// ============================================
// DB_RecipeProgram1 - Program 1
// Lines: 500
// CHUNKS: 5 x 100
// Generated by SpinningCam  [2026-09-24 16:45:37]
// !!! CONTINUOUS MOTION (CMD=2) - EXPERIMENTAL PLC ONLY !!!
// Load ONLY on the continuous-motion PLC build. A production PLC
// skips CMD=2 lines and jumps straight between the other points.
// T=0.045 s, corner tol=0.2 mm, F min=180, exact stop at >= 90 deg, stop slow-down=OFF
// CMD=2 lines: 483, exact corners: 2, slowed corners: 1 (+1 leaving), slowed stops: 0
// ============================================
//
// --- MAKINE AYARLARI ---
// Machine Origin  : X=0.0, Z=0.0
// Axis Direction  : X=NORMAL, Z=NORMAL
// Output Mode     : RADIUS
// G54 Offset      : X=0.0, Z=0.0
// Home            : X=-394.0, Z=-174.0
// Retract         : X=-10.0, Z=-10.0
//
// --- PARCA / BLANK ---
// Blank Radius    : 150.0 mm
// Blank Z Shift   : 0.0 mm
// Final Thickness : 0.8 mm
// Min Safety Gap  : 0.0 mm
//
// --- MANDREL POZISYON ---
// Mandrel Offset  : X=0.0, Z=0.0
// Mandrel Rot     : Rx=90.0, Ry=0.0, Rz=0.0
//
// --- OPERASYONLAR ---
// Op1: ROUGHING, 1 paso, T004, R=44.56mm, RPM=600.0, mm_min=1000.0
// Op2: ROUGHING, 1 paso, T004, R=44.56mm, RPM=600.0, mm_min=1000.0
// Op3: ROUGHING, 1 paso, T004, R=44.56mm, RPM=600.0, mm_min=1000.0
// Op4: ROUGHING, 1 paso, T004, R=44.56mm, RPM=600.0, mm_min=1000.0
// Op5: ROUGHING, 1 paso, T004, R=44.56mm, RPM=600.0, mm_min=1000.0
// Op6: ROUGHING, 1 paso, T004, R=44.56mm, RPM=600.0, mm_min=1000.0
// Op7: ROUGHING, 1 paso, T004, R=44.56mm, RPM=600.0, mm_min=1000.0
// Op8: ROUGHING, 1 paso, T004, R=44.56mm, RPM=600.0, mm_min=1000.0
// Op9: ROUGHING, 1 paso, T004, R=44.56mm, RPM=600.0, mm_min=1000.0
// Op10: ROUGHING, 1 paso, T004, R=44.56mm, RPM=600.0, mm_min=1000.0
// Op11: ROUGHING, 1 paso, T004, R=44.56mm, RPM=600.0, mm_min=1000.0
// Op12: ROUGHING, 1 paso, T004, R=44.56mm, RPM=600.0, mm_min=1000.0
// Op13: ROUGHING, 1 paso, T004, R=44.56mm, RPM=600.0, mm_min=1000.0
// Op14: ROUGHING, 1 paso, T004, R=44.56mm, RPM=600.0, mm_min=1000.0
// Op15: ROUGHING, 1 paso, T004, R=44.56mm, RPM=600.0, mm_min=1000.0
// Op16: ROUGHING, 1 paso, T004, R=44.56mm, RPM=600.0, mm_min=1000.0
// Op17: ROUGHING, 1 paso, T004, R=44.56mm, RPM=600.0, mm_min=1000.0
// Op18: CUTTING, 1 paso, T006, R=5.0mm, RPM=500.0, mm_min=7.0
// Op19: ROUGHING, 1 paso, T004, R=44.56mm, RPM=600.0, mm_min=1000.0
// Op20: ROUGHING, 1 paso, T004, R=44.56mm, RPM=600.0, mm_min=1000.0
// Op21: ROUGHING, 1 paso, T004, R=44.56mm, RPM=600.0, mm_min=1000.0
// Op22: ROUGHING, 1 paso, T004, R=44.56mm, RPM=600.0, mm_min=1000.0
// Op23: ROUGHING, 1 paso, T004, R=44.56mm, RPM=600.0, mm_min=1000.0
// Op24: ROUGHING, 1 paso, T004, R=44.56mm, RPM=600.0, mm_min=1000.0
// Op25: ROUGHING, 1 paso, T004, R=44.56mm, RPM=600.0, mm_min=1000.0
// Op26: ROUGHING, 1 paso, T004, R=44.56mm, RPM=600.0, mm_min=1000.0
// Op27: ROUGHING, 1 paso, T004, R=44.56mm, RPM=600.0, mm_min=1000.0
// Op28: ROUGHING, 1 paso, T004, R=44.56mm, RPM=600.0, mm_min=1000.0
// Op29: ROUGHING, 1 paso, T004, R=44.56mm, RPM=600.0, mm_min=1000.0
// Op30: ROUGHING, 1 paso, T004, R=44.56mm, RPM=600.0, mm_min=1000.0
// Op31: ROUGHING, 1 paso, T004, R=44.56mm, RPM=600.0, mm_min=1000.0
// Op32: ROUGHING, 1 paso, T004, R=44.56mm, RPM=600.0, mm_min=1000.0
// Op33: ROUGHING, 1 paso, T004, R=44.56mm, RPM=600.0, mm_min=1000.0
// Op34: ROUGHING, 1 paso, T004, R=44.56mm, RPM=600.0, mm_min=1000.0
// Op35: ROUGHING, 1 paso, T004, R=44.56mm, RPM=600.0, mm_min=1000.0
// Op36: ROUGHING, 1 paso, T004, R=44.56mm, RPM=600.0, mm_min=1000.0
// Op37: ROUGHING, 1 paso, T004, R=44.56mm, RPM=600.0, mm_min=1000.0
// Op38: ROUGHING, 1 paso, T004, R=44.56mm, RPM=600.0, mm_min=1000.0
// Op39: ROUGHING, 1 paso, T004, R=44.56mm, RPM=600.0, mm_min=1000.0
// Op40: ROUGHING, 1 paso, T004, R=44.56mm, RPM=600.0, mm_min=1000.0
// Op41: ROUGHING, 1 paso, T004, R=44.56mm, RPM=600.0, mm_min=1000.0
// Op42: ROUGHING, 1 paso, T004, R=44.56mm, RPM=600.0, mm_min=1000.0
// Op43: ROUGHING, 1 paso, T004, R=44.56mm, RPM=600.0, mm_min=1000.0
// Op44: ROUGHING, 1 paso, T004, R=44.56mm, RPM=600.0, mm_min=1000.0
// Op45: ROUGHING, 1 paso, T004, R=44.56mm, RPM=600.0, mm_min=1000.0
// Op46: ROUGHING, 1 paso, T004, R=44.56mm, RPM=600.0, mm_min=1000.0
// Op47: ROUGHING, 1 paso, T004, R=44.56mm, RPM=600.0, mm_min=1000.0
// Op48: ROUGHING, 1 paso, T004, R=44.56mm, RPM=600.0, mm_min=1000.0
// Op49: ROUGHING, 1 paso, T004, R=44.56mm, RPM=600.0, mm_min=1000.0
// Op50: ROUGHING, 1 paso, T004, R=44.56mm, RPM=600.0, mm_min=1000.0
// Op51: ROUGHING, 1 paso, T004, R=44.56mm, RPM=600.0, mm_min=1000.0
// Op52: ROUGHING, 1 paso, T004, R=44.56mm, RPM=600.0, mm_min=1000.0
// Op53: ROUGHING, 1 paso, T004, R=44.56mm, RPM=600.0, mm_min=1000.0
// Op54: ROUGHING, 1 paso, T004, R=44.56mm, RPM=600.0, mm_min=1000.0
// Op55: ROUGHING, 1 paso, T004, R=44.56mm, RPM=600.0, mm_min=1000.0
// Op56: ROUGHING, 1 paso, T004, R=44.56mm, RPM=600.0, mm_min=1000.0
// Op57: ROUGHING, 1 paso, T004, R=44.56mm, RPM=600.0, mm_min=1000.0
// Op58: ROUGHING, 1 paso, T004, R=44.56mm, RPM=600.0, mm_min=1000.0
// Op59: ROUGHING, 1 paso, T004, R=44.56mm, RPM=600.0, mm_min=1000.0
// Op60: ROUGHING, 1 paso, T004, R=44.56mm, RPM=600.0, mm_min=1000.0
// Op61: ROUGHING, 1 paso, T004, R=44.56mm, RPM=600.0, mm_min=1000.0
// Op62: ROUGHING, 1 paso, T004, R=44.56mm, RPM=600.0, mm_min=1000.0
// Op63: ROUGHING, 1 paso, T004, R=44.56mm, RPM=600.0, mm_min=1000.0
// Op64: ROUGHING, 1 paso, T004, R=44.56mm, RPM=600.0, mm_min=1000.0
// Op65: ROUGHING, 1 paso, T004, R=44.56mm, RPM=600.0, mm_min=1000.0
// Op66: ROUGHING, 1 paso, T004, R=44.56mm, RPM=600.0, mm_min=1000.0
// Op67: ROUGHING, 1 paso, T004, R=44.56mm, RPM=600.0, mm_min=1000.0
// Op68: ROUGHING, 1 paso, T004, R=44.56mm, RPM=600.0, mm_min=1000.0
// Op69: ROUGHING, 1 paso, T004, R=44.56mm, RPM=600.0, mm_min=1000.0
// Op70: ROUGHING, 1 paso, T004, R=44.56mm, RPM=600.0, mm_min=1000.0
// Op71: ROUGHING, 1 paso, T004, R=44.56mm, RPM=600.0, mm_min=1000.0
// Op72: ROUGHING, 1 paso, T004, R=44.56mm, RPM=600.0, mm_min=1000.0
// Op73: ROUGHING, 1 paso, T004, R=44.56mm, RPM=600.0, mm_min=1000.0
// Op74: ROUGHING, 1 paso, T004, R=44.56mm, RPM=600.0, mm_min=1000.0
// Op75: ROUGHING, 1 paso, T004, R=44.56mm, RPM=600.0, mm_min=1000.0
// Op76: ROUGHING, 1 paso, T004, R=44.56mm, RPM=600.0, mm_min=1000.0
// Op77: ROUGHING, 1 paso, T004, R=44.56mm, RPM=600.0, mm_min=1000.0
// Op78: ROUGHING, 1 paso, T004, R=44.56mm, RPM=600.0, mm_min=1000.0
// Op79: ROUGHING, 1 paso, T004, R=44.56mm, RPM=600.0, mm_min=1000.0
// Op80: ROUGHING, 1 paso, T004, R=44.56mm, RPM=600.0, mm_min=1000.0
// Op81: ROUGHING, 1 paso, T004, R=44.56mm, RPM=600.0, mm_min=1000.0
// Op82: ROUGHING, 1 paso, T004, R=44.56mm, RPM=600.0, mm_min=1000.0
// Op83: ROUGHING, 1 paso, T004, R=44.56mm, RPM=600.0, mm_min=1000.0
// Op84: ROUGHING, 1 paso, T004, R=44.56mm, RPM=600.0, mm_min=1000.0
// Op85: ROUGHING, 1 paso, T004, R=44.56mm, RPM=600.0, mm_min=1000.0
// Op86: ROUGHING, 1 paso, T004, R=44.56mm, RPM=600.0, mm_min=1000.0
// Op87: ROUGHING, 1 paso, T004, R=44.56mm, RPM=600.0, mm_min=1000.0
// Op88: ROUGHING, 1 paso, T004, R=44.56mm, RPM=600.0, mm_min=1000.0
// Op89: ROUGHING, 1 paso, T004, R=44.56mm, RPM=600.0, mm_min=1000.0
// Op90: ROUGHING, 1 paso, T004, R=44.56mm, RPM=600.0, mm_min=1000.0
// Op91: ROUGHING, 1 paso, T004, R=44.56mm, RPM=600.0, mm_min=1000.0
// Op92: ROUGHING, 1 paso, T004, R=44.56mm, RPM=600.0, mm_min=1000.0
// Op93: ROUGHING, 1 paso, T004, R=44.56mm, RPM=600.0, mm_min=1000.0
// Op94: ROUGHING, 1 paso, T004, R=44.56mm, RPM=600.0, mm_min=1000.0
// Op95: ROUGHING, 1 paso, T004, R=44.56mm, RPM=600.0, mm_min=1000.0
// Op96: ROUGHING, 1 paso, T004, R=44.56mm, RPM=600.0, mm_min=1000.0
// Op97: ROUGHING, 1 paso, T004, R=44.56mm, RPM=600.0, mm_min=1000.0
// Op98: ROUGHING, 1 paso, T004, R=44.56mm, RPM=600.0, mm_min=1000.0
// Op99: ROUGHING, 1 paso, T004, R=44.56mm, RPM=600.0, mm_min=1000.0
// Op100: ROUGHING, 1 paso, T004, R=44.56mm, RPM=600.0, mm_min=1000.0
// Op101: ROUGHING, 1 paso, T004, R=44.56mm, RPM=600.0, mm_min=1000.0
// Op102: ROUGHING, 1 paso, T004, R=44.56mm, RPM=600.0, mm_min=1000.0
// Op103: ROUGHING, 1 paso, T004, R=44.56mm, RPM=600.0, mm_min=1000.0
// Op104: ROUGHING, 1 paso, T004, R=44.56mm, RPM=600.0, mm_min=1000.0
// Op105: ROUGHING, 1 paso, T004, R=44.56mm, RPM=600.0, mm_min=1000.0
// Op106: ROUGHING, 1 paso, T004, R=44.56mm, RPM=600.0, mm_min=1000.0
// Op107: ROUGHING, 1 paso, T004, R=44.56mm, RPM=600.0, mm_min=1000.0
// Op108: ROUGHING, 1 paso, T004, R=44.56mm, RPM=600.0, mm_min=1000.0
// Op109: ROUGHING, 1 paso, T004, R=44.56mm, RPM=600.0, mm_min=1000.0
// Op110: ROUGHING, 1 paso, T004, R=44.56mm, RPM=600.0, mm_min=1000.0
// Op111: ROUGHING, 1 paso, T004, R=44.56mm, RPM=600.0, mm_min=1000.0
// Op112: ROUGHING, 1 paso, T004, R=44.56mm, RPM=600.0, mm_min=1000.0
// Op113: CUTTING, 1 paso, T006, R=5.0mm, RPM=500.0, mm_min=7.0
// Op114: ROUGHING, 1 paso, T004, R=44.56mm, RPM=600.0, mm_min=1000.0
// Op115: ROUGHING, 1 paso, T004, R=44.56mm, RPM=600.0, mm_min=1000.0
// Op116: ROUGHING, 1 paso, T004, R=44.56mm, RPM=600.0, mm_min=1000.0
// Op117: ROUGHING, 1 paso, T004, R=44.56mm, RPM=600.0, mm_min=1000.0
// Op118: ROUGHING, 1 paso, T004, R=44.56mm, RPM=600.0, mm_min=1000.0
// Op119: ROUGHING, 1 paso, T004, R=44.56mm, RPM=600.0, mm_min=1000.0
// Op120: ROUGHING, 1 paso, T004, R=44.56mm, RPM=600.0, mm_min=1000.0
// Op121: ROUGHING, 1 paso, T004, R=44.56mm, RPM=600.0, mm_min=400.0
// Op122: ROUGHING, 1 paso, T004, R=44.56mm, RPM=600.0, mm_min=400.0
// Op123: ROUGHING, 1 paso, T004, R=44.56mm, RPM=600.0, mm_min=400.0
// Op124: ROUGHING, 1 paso, T004, R=44.56mm, RPM=600.0, mm_min=1000.0
// Op125: ROUGHING, 1 paso, T004, R=44.56mm, RPM=600.0, mm_min=400.0
// Op126: ROUGHING, 1 paso, T004, R=44.56mm, RPM=600.0, mm_min=400.0
// Op127: ROUGHING, 1 paso, T004, R=44.56mm, RPM=600.0, mm_min=400.0
// Op128: ROUGHING, 1 paso, T004, R=44.56mm, RPM=600.0, mm_min=400.0
// Op129: ROUGHING, 1 paso, T004, R=44.56mm, RPM=600.0, mm_min=400.0
// Op130: ROUGHING, 1 paso, T004, R=44.56mm, RPM=600.0, mm_min=400.0
// Op131: ROUGHING, 1 paso, T004, R=44.56mm, RPM=600.0, mm_min=400.0
// Op132: ROUGHING, 1 paso, T004, R=44.56mm, RPM=600.0, mm_min=400.0
// Op133: ROUGHING, 1 paso, T004, R=44.56mm, RPM=600.0, mm_min=400.0
// Op134: ROUGHING, 1 paso, T004, R=44.56mm, RPM=600.0, mm_min=400.0
// Op135: ROUGHING, 1 paso, T004, R=44.56mm, RPM=600.0, mm_min=400.0
// Op136: ROUGHING, 1 paso, T004, R=44.56mm, RPM=600.0, mm_min=400.0
// Op137: ROUGHING, 1 paso, T004, R=44.56mm, RPM=600.0, mm_min=400.0
// Op138: ROUGHING, 1 paso, T004, R=44.56mm, RPM=600.0, mm_min=400.0
// Op139: ROUGHING, 1 paso, T004, R=44.56mm, RPM=600.0, mm_min=400.0
// Op140: ROUGHING, 1 paso, T004, R=44.56mm, RPM=600.0, mm_min=400.0
// Op141: ROUGHING, 1 paso, T004, R=44.56mm, RPM=600.0, mm_min=400.0
// Op142: ROUGHING, 1 paso, T004, R=44.56mm, RPM=600.0, mm_min=400.0
// Op143: ROUGHING, 1 paso, T004, R=44.56mm, RPM=600.0, mm_min=400.0
// Op144: ROUGHING, 1 paso, T004, R=44.56mm, RPM=600.0, mm_min=400.0
// Op145: ROUGHING, 1 paso, T004, R=44.56mm, RPM=600.0, mm_min=400.0
// Op146: ROUGHING, 1 paso, T004, R=44.56mm, RPM=600.0, mm_min=400.0
// Op147: ROUGHING, 1 paso, T004, R=44.56mm, RPM=600.0, mm_min=400.0
// Op148: ROUGHING, 1 paso, T004, R=44.56mm, RPM=600.0, mm_min=400.0
// Op149: ROUGHING, 1 paso, T004, R=44.56mm, RPM=600.0, mm_min=400.0
// Op150: ROUGHING, 1 paso, T004, R=44.56mm, RPM=600.0, mm_min=400.0
// Op151: ROUGHING, 1 paso, T004, R=44.56mm, RPM=800.0, mm_min=400.0
// Op152: ROUGHING, 1 paso, T004, R=44.56mm, RPM=800.0, mm_min=400.0
// Op153: ROUGHING, 1 paso, T004, R=44.56mm, RPM=800.0, mm_min=400.0
// Op154: ROUGHING, 1 paso, T004, R=44.56mm, RPM=800.0, mm_min=400.0
// Op155: ROUGHING, 1 paso, T004, R=44.56mm, RPM=800.0, mm_min=400.0
// Op156: ROUGHING, 1 paso, T004, R=44.56mm, RPM=800.0, mm_min=400.0
// Op157: ROUGHING, 1 paso, T004, R=44.56mm, RPM=800.0, mm_min=400.0
// Op158: ROUGHING, 1 paso, T004, R=44.56mm, RPM=800.0, mm_min=400.0
// Op159: ROUGHING, 1 paso, T004, R=44.56mm, RPM=800.0, mm_min=400.0
// Op160: ROUGHING, 1 paso, T004, R=44.56mm, RPM=800.0, mm_min=400.0
// Op161: ROUGHING, 1 paso, T004, R=44.56mm, RPM=800.0, mm_min=400.0
// Op162: ROUGHING, 1 paso, T004, R=44.56mm, RPM=800.0, mm_min=400.0
// Op163: ROUGHING, 1 paso, T004, R=44.56mm, RPM=800.0, mm_min=400.0
// Op164: ROUGHING, 1 paso, T004, R=44.56mm, RPM=800.0, mm_min=400.0
// Op165: ROUGHING, 1 paso, T004, R=44.56mm, RPM=800.0, mm_min=400.0
// Op166: ROUGHING, 1 paso, T004, R=44.56mm, RPM=800.0, mm_min=400.0
// Op167: ROUGHING, 1 paso, T004, R=44.56mm, RPM=800.0, mm_min=400.0
// ============================================

DATA_BLOCK "DB_RecipeProgram1"
{ S7_Optimized_Access := 'FALSE' }
VERSION : 0.2
UNLINKED
NON_RETAIN
    VAR
        Header : "RecipeHeader";
        Lines1 : Array[0..99] of "RecipeLine";  // global lines 0..99
        Lines2 : Array[0..99] of "RecipeLine";  // global lines 100..199
        Lines3 : Array[0..99] of "RecipeLine";  // global lines 200..299
        Lines4 : Array[0..99] of "RecipeLine";  // global lines 300..399
        Lines5 : Array[0..99] of "RecipeLine";  // global lines 400..499
    END_VAR
BEGIN
    // Header
    Header.sName := 'Program 1';
    Header.LineCount := 500;
    Header.Valid := TRUE;
    Header.PreScanned := FALSE;
    Header.MinX := 174.000;
    Header.MaxX := 273.136;
    Header.MinZ := 74.000;
    Header.MaxZ := 374.142;

    // --- Tool table (CAM-authored) ---
    Header.ProvidesToolConfig := TRUE;
    Header.ToolCount := 4;
    Header.AutoCalcAngles := FALSE;
    Header.ToolCode_List[1] := 4;
    Header.ToolCode_List[2] := 5;
    Header.ToolCode_List[3] := 6;
    Header.ToolCode_List[4] := 7;
    Header.ToolAngle_List[1] := 0.0;
    Header.ToolAngle_List[2] := 120.0;
    Header.ToolAngle_List[3] := 240.0;
    Header.ToolAngle_List[4] := 360.0;

    // --- Integrity ---
    // Order-sensitive sum over CMD+Param+F of lines 0..LineCount-1.
    // The PLC recomputes it after reassembling the chunks and refuses
    // to run on a mismatch (16#0316). X/Z are excluded on purpose:
    // float32-vs-float64 rounding would eventually cry wolf.
    Header.ProvidesChecksum := TRUE;
    Header.Checksum := 121162007;

    // Recipe Lines (500 total)

    // --- Lines1 (global lines 0..99) ---
    Lines1[0].X := 0.000; Lines1[0].Z := 0.000; Lines1[0].F := 0; Lines1[0].CMD := 40; Lines1[0].Param := 80; // Cylinder GOTO P80
    Lines1[1].X := 0.000; Lines1[1].Z := 0.000; Lines1[1].F := 0; Lines1[1].CMD := 10; Lines1[1].Param := 4; // Tool Change T4
    Lines1[2].X := 0.000; Lines1[2].Z := 0.000; Lines1[2].F := 0; Lines1[2].CMD := 20; Lines1[2].Param := 60; // Spindle ON 600 RPM
    Lines1[3].X := 0.000; Lines1[3].Z := 0.000; Lines1[3].F := 0; Lines1[3].CMD := 41; Lines1[3].Param := 1; // M41 (Clamp On) P1 [Op67 P1]
    Lines1[4].X := 259.077; Lines1[4].Z := 181.006; Lines1[4].F := 0; Lines1[4].CMD := 0; Lines1[4].Param := 0; // G0 Rapid [Op67 P1]
    Lines1[5].X := 259.982; Lines1[5].Z := 183.614; Lines1[5].F := 1000; Lines1[5].CMD := 2; Lines1[5].Param := 0; // G1 Continuous [Op67 P1]
    Lines1[6].X := 260.781; Lines1[6].Z := 186.001; Lines1[6].F := 1000; Lines1[6].CMD := 2; Lines1[6].Param := 0; // G1 Continuous [Op67 P1]
    Lines1[7].X := 261.558; Lines1[7].Z := 188.404; Lines1[7].F := 1000; Lines1[7].CMD := 2; Lines1[7].Param := 0; // G1 Continuous [Op67 P1]
    Lines1[8].X := 262.311; Lines1[8].Z := 190.820; Lines1[8].F := 1000; Lines1[8].CMD := 2; Lines1[8].Param := 0; // G1 Continuous [Op67 P1]
    Lines1[9].X := 263.113; Lines1[9].Z := 193.493; Lines1[9].F := 1000; Lines1[9].CMD := 2; Lines1[9].Param := 0; // G1 Continuous [Op67 P1]
    Lines1[10].X := 263.818; Lines1[10].Z := 195.938; Lines1[10].F := 1000; Lines1[10].CMD := 2; Lines1[10].Param := 0; // G1 Continuous [Op67 P1]
    Lines1[11].X := 264.498; Lines1[11].Z := 198.394; Lines1[11].F := 1000; Lines1[11].CMD := 2; Lines1[11].Param := 0; // G1 Continuous [Op67 P1]
    Lines1[12].X := 265.155; Lines1[12].Z := 200.863; Lines1[12].F := 1000; Lines1[12].CMD := 2; Lines1[12].Param := 0; // G1 Continuous [Op67 P1]
    Lines1[13].X := 265.850; Lines1[13].Z := 203.592; Lines1[13].F := 1000; Lines1[13].CMD := 2; Lines1[13].Param := 0; // G1 Continuous [Op67 P1]
    Lines1[14].X := 266.456; Lines1[14].Z := 206.084; Lines1[14].F := 1000; Lines1[14].CMD := 2; Lines1[14].Param := 0; // G1 Continuous [Op67 P1]
    Lines1[15].X := 267.037; Lines1[15].Z := 208.586; Lines1[15].F := 1000; Lines1[15].CMD := 2; Lines1[15].Param := 0; // G1 Continuous [Op67 P1]
    Lines1[16].X := 267.593; Lines1[16].Z := 211.098; Lines1[16].F := 1000; Lines1[16].CMD := 2; Lines1[16].Param := 0; // G1 Continuous [Op67 P1]
    Lines1[17].X := 268.125; Lines1[17].Z := 213.620; Lines1[17].F := 1000; Lines1[17].CMD := 2; Lines1[17].Param := 0; // G1 Continuous [Op67 P1]
    Lines1[18].X := 268.631; Lines1[18].Z := 216.150; Lines1[18].F := 1000; Lines1[18].CMD := 2; Lines1[18].Param := 0; // G1 Continuous [Op67 P1]
    Lines1[19].X := 269.111; Lines1[19].Z := 218.688; Lines1[19].F := 1000; Lines1[19].CMD := 2; Lines1[19].Param := 0; // G1 Continuous [Op67 P1]
    Lines1[20].X := 269.566; Lines1[20].Z := 221.233; Lines1[20].F := 1000; Lines1[20].CMD := 2; Lines1[20].Param := 0; // G1 Continuous [Op67 P1]
    Lines1[21].X := 269.994; Lines1[21].Z := 223.786; Lines1[21].F := 1000; Lines1[21].CMD := 2; Lines1[21].Param := 0; // G1 Continuous [Op67 P1]
    Lines1[22].X := 270.396; Lines1[22].Z := 226.346; Lines1[22].F := 1000; Lines1[22].CMD := 2; Lines1[22].Param := 0; // G1 Continuous [Op67 P1]
    Lines1[23].X := 270.772; Lines1[23].Z := 228.911; Lines1[23].F := 1000; Lines1[23].CMD := 2; Lines1[23].Param := 0; // G1 Continuous [Op67 P1]
    Lines1[24].X := 271.121; Lines1[24].Z := 231.482; Lines1[24].F := 1000; Lines1[24].CMD := 2; Lines1[24].Param := 0; // G1 Continuous [Op67 P1]
    Lines1[25].X := 271.443; Lines1[25].Z := 234.057; Lines1[25].F := 1000; Lines1[25].CMD := 2; Lines1[25].Param := 0; // G1 Continuous [Op67 P1]
    Lines1[26].X := 271.737; Lines1[26].Z := 236.638; Lines1[26].F := 1000; Lines1[26].CMD := 2; Lines1[26].Param := 0; // G1 Continuous [Op67 P1]
    Lines1[27].X := 272.005; Lines1[27].Z := 239.222; Lines1[27].F := 1000; Lines1[27].CMD := 2; Lines1[27].Param := 0; // G1 Continuous [Op67 P1]
    Lines1[28].X := 272.244; Lines1[28].Z := 241.809; Lines1[28].F := 1000; Lines1[28].CMD := 2; Lines1[28].Param := 0; // G1 Continuous [Op67 P1]
    Lines1[29].X := 272.456; Lines1[29].Z := 244.399; Lines1[29].F := 1000; Lines1[29].CMD := 2; Lines1[29].Param := 0; // G1 Continuous [Op67 P1]
    Lines1[30].X := 272.639; Lines1[30].Z := 246.991; Lines1[30].F := 1000; Lines1[30].CMD := 2; Lines1[30].Param := 0; // G1 Continuous [Op67 P1]
    Lines1[31].X := 272.794; Lines1[31].Z := 249.585; Lines1[31].F := 1000; Lines1[31].CMD := 2; Lines1[31].Param := 0; // G1 Continuous [Op67 P1]
    Lines1[32].X := 272.910; Lines1[32].Z := 251.921; Lines1[32].F := 1000; Lines1[32].CMD := 2; Lines1[32].Param := 0; // G1 Continuous [Op67 P1]
    Lines1[33].X := 273.010; Lines1[33].Z := 254.517; Lines1[33].F := 1000; Lines1[33].CMD := 2; Lines1[33].Param := 0; // G1 Continuous [Op67 P1]
    Lines1[34].X := 273.081; Lines1[34].Z := 257.112; Lines1[34].F := 1000; Lines1[34].CMD := 2; Lines1[34].Param := 0; // G1 Continuous [Op67 P1]
    Lines1[35].X := 273.124; Lines1[35].Z := 259.708; Lines1[35].F := 1000; Lines1[35].CMD := 2; Lines1[35].Param := 0; // G1 Continuous [Op67 P1]
    Lines1[36].X := 273.136; Lines1[36].Z := 262.043; Lines1[36].F := 1000; Lines1[36].CMD := 2; Lines1[36].Param := 0; // G1 Continuous [Op67 P1]
    Lines1[37].X := 273.127; Lines1[37].Z := 264.118; Lines1[37].F := 1000; Lines1[37].CMD := 2; Lines1[37].Param := 0; // G1 Continuous [Op67 P1]
    Lines1[38].X := 273.099; Lines1[38].Z := 266.192; Lines1[38].F := 1000; Lines1[38].CMD := 2; Lines1[38].Param := 0; // G1 Continuous [Op67 P1]
    Lines1[39].X := 272.994; Lines1[39].Z := 270.075; Lines1[39].F := 1000; Lines1[39].CMD := 2; Lines1[39].Param := 0; // G1 Continuous [Op67 P1]
    Lines1[40].X := 272.910; Lines1[40].Z := 272.144; Lines1[40].F := 1000; Lines1[40].CMD := 2; Lines1[40].Param := 0; // G1 Continuous [Op67 P1]
    Lines1[41].X := 272.807; Lines1[41].Z := 274.211; Lines1[41].F := 1000; Lines1[41].CMD := 2; Lines1[41].Param := 0; // G1 Continuous [Op67 P1]
    Lines1[42].X := 272.684; Lines1[42].Z := 276.274; Lines1[42].F := 1000; Lines1[42].CMD := 2; Lines1[42].Param := 0; // G1 Continuous [Op67 P1]
    Lines1[43].X := 272.559; Lines1[43].Z := 278.078; Lines1[43].F := 1000; Lines1[43].CMD := 2; Lines1[43].Param := 0; // G1 Continuous [Op67 P1]
    Lines1[44].X := 272.399; Lines1[44].Z := 280.137; Lines1[44].F := 1000; Lines1[44].CMD := 2; Lines1[44].Param := 0; // G1 Continuous [Op67 P1]
    Lines1[45].X := 272.242; Lines1[45].Z := 281.935; Lines1[45].F := 1000; Lines1[45].CMD := 2; Lines1[45].Param := 0; // G1 Continuous [Op67 P1]
    Lines1[46].X := 272.043; Lines1[46].Z := 283.987; Lines1[46].F := 1000; Lines1[46].CMD := 2; Lines1[46].Param := 0; // G1 Continuous [Op67 P1]
    Lines1[47].X := 271.853; Lines1[47].Z := 285.780; Lines1[47].F := 1000; Lines1[47].CMD := 2; Lines1[47].Param := 0; // G1 Continuous [Op67 P1]
    Lines1[48].X := 271.617; Lines1[48].Z := 287.824; Lines1[48].F := 1000; Lines1[48].CMD := 2; Lines1[48].Param := 0; // G1 Continuous [Op67 P1]
    Lines1[49].X := 271.393; Lines1[49].Z := 289.610; Lines1[49].F := 1000; Lines1[49].CMD := 2; Lines1[49].Param := 0; // G1 Continuous [Op67 P1]
    Lines1[50].X := 271.118; Lines1[50].Z := 291.646; Lines1[50].F := 1000; Lines1[50].CMD := 2; Lines1[50].Param := 0; // G1 Continuous [Op67 P1]
    Lines1[51].X := 270.860; Lines1[51].Z := 293.424; Lines1[51].F := 1000; Lines1[51].CMD := 2; Lines1[51].Param := 0; // G1 Continuous [Op67 P1]
    Lines1[52].X := 270.545; Lines1[52].Z := 295.451; Lines1[52].F := 1000; Lines1[52].CMD := 2; Lines1[52].Param := 0; // G1 Continuous [Op67 P1]
    Lines1[53].X := 270.253; Lines1[53].Z := 297.220; Lines1[53].F := 1000; Lines1[53].CMD := 2; Lines1[53].Param := 0; // G1 Continuous [Op67 P1]
    Lines1[54].X := 269.900; Lines1[54].Z := 299.237; Lines1[54].F := 1000; Lines1[54].CMD := 2; Lines1[54].Param := 0; // G1 Continuous [Op67 P1]
    Lines1[55].X := 269.573; Lines1[55].Z := 300.996; Lines1[55].F := 1000; Lines1[55].CMD := 2; Lines1[55].Param := 0; // G1 Continuous [Op67 P1]
    Lines1[56].X := 269.179; Lines1[56].Z := 303.002; Lines1[56].F := 1000; Lines1[56].CMD := 2; Lines1[56].Param := 0; // G1 Continuous [Op67 P1]
    Lines1[57].X := 268.817; Lines1[57].Z := 304.751; Lines1[57].F := 1000; Lines1[57].CMD := 2; Lines1[57].Param := 0; // G1 Continuous [Op67 P1]
    Lines1[58].X := 268.383; Lines1[58].Z := 306.745; Lines1[58].F := 1000; Lines1[58].CMD := 2; Lines1[58].Param := 0; // G1 Continuous [Op67 P1]
    Lines1[59].X := 267.986; Lines1[59].Z := 308.483; Lines1[59].F := 1000; Lines1[59].CMD := 2; Lines1[59].Param := 0; // G1 Continuous [Op67 P1]
    Lines1[60].X := 267.511; Lines1[60].Z := 310.463; Lines1[60].F := 1000; Lines1[60].CMD := 2; Lines1[60].Param := 0; // G1 Continuous [Op67 P1]
    Lines1[61].X := 267.078; Lines1[61].Z := 312.190; Lines1[61].F := 1000; Lines1[61].CMD := 2; Lines1[61].Param := 0; // G1 Continuous [Op67 P1]
    Lines1[62].X := 266.628; Lines1[62].Z := 313.910; Lines1[62].F := 1000; Lines1[62].CMD := 2; Lines1[62].Param := 0; // G1 Continuous [Op67 P1]
    Lines1[63].X := 266.161; Lines1[63].Z := 315.625; Lines1[63].F := 1000; Lines1[63].CMD := 2; Lines1[63].Param := 0; // G1 Continuous [Op67 P1]
    Lines1[64].X := 265.607; Lines1[64].Z := 317.576; Lines1[64].F := 1000; Lines1[64].CMD := 2; Lines1[64].Param := 0; // G1 Continuous [Op67 P1]
    Lines1[65].X := 265.103; Lines1[65].Z := 319.277; Lines1[65].F := 1000; Lines1[65].CMD := 2; Lines1[65].Param := 0; // G1 Continuous [Op67 P1]
    Lines1[66].X := 264.582; Lines1[66].Z := 320.972; Lines1[66].F := 1000; Lines1[66].CMD := 2; Lines1[66].Param := 0; // G1 Continuous [Op67 P1]
    Lines1[67].X := 264.045; Lines1[67].Z := 322.659; Lines1[67].F := 1000; Lines1[67].CMD := 2; Lines1[67].Param := 0; // G1 Continuous [Op67 P1]
    Lines1[68].X := 263.489; Lines1[68].Z := 324.339; Lines1[68].F := 1000; Lines1[68].CMD := 2; Lines1[68].Param := 0; // G1 Continuous [Op67 P1]
    Lines1[69].X := 262.917; Lines1[69].Z := 326.013; Lines1[69].F := 1000; Lines1[69].CMD := 2; Lines1[69].Param := 0; // G1 Continuous [Op67 P1]
    Lines1[70].X := 262.326; Lines1[70].Z := 327.679; Lines1[70].F := 1000; Lines1[70].CMD := 2; Lines1[70].Param := 0; // G1 Continuous [Op67 P1]
    Lines1[71].X := 261.719; Lines1[71].Z := 329.337; Lines1[71].F := 1000; Lines1[71].CMD := 2; Lines1[71].Param := 0; // G1 Continuous [Op67 P1]
    Lines1[72].X := 261.093; Lines1[72].Z := 330.988; Lines1[72].F := 1000; Lines1[72].CMD := 2; Lines1[72].Param := 0; // G1 Continuous [Op67 P1]
    Lines1[73].X := 260.450; Lines1[73].Z := 332.630; Lines1[73].F := 1000; Lines1[73].CMD := 2; Lines1[73].Param := 0; // G1 Continuous [Op67 P1]
    Lines1[74].X := 259.789; Lines1[74].Z := 334.265; Lines1[74].F := 1000; Lines1[74].CMD := 2; Lines1[74].Param := 0; // G1 Continuous [Op67 P1]
    Lines1[75].X := 259.110; Lines1[75].Z := 335.891; Lines1[75].F := 1000; Lines1[75].CMD := 2; Lines1[75].Param := 0; // G1 Continuous [Op67 P1]
    Lines1[76].X := 258.413; Lines1[76].Z := 337.509; Lines1[76].F := 1000; Lines1[76].CMD := 2; Lines1[76].Param := 0; // G1 Continuous [Op67 P1]
    Lines1[77].X := 257.699; Lines1[77].Z := 339.118; Lines1[77].F := 1000; Lines1[77].CMD := 2; Lines1[77].Param := 0; // G1 Continuous [Op67 P1]
    Lines1[78].X := 256.966; Lines1[78].Z := 340.718; Lines1[78].F := 1000; Lines1[78].CMD := 2; Lines1[78].Param := 0; // G1 Continuous [Op67 P1]
    Lines1[79].X := 256.215; Lines1[79].Z := 342.310; Lines1[79].F := 1000; Lines1[79].CMD := 2; Lines1[79].Param := 0; // G1 Continuous [Op67 P1]
    Lines1[80].X := 255.447; Lines1[80].Z := 343.893; Lines1[80].F := 1000; Lines1[80].CMD := 2; Lines1[80].Param := 0; // G1 Continuous [Op67 P1]
    Lines1[81].X := 254.662; Lines1[81].Z := 345.467; Lines1[81].F := 1000; Lines1[81].CMD := 2; Lines1[81].Param := 0; // G1 Continuous [Op67 P1]
    Lines1[82].X := 253.860; Lines1[82].Z := 347.032; Lines1[82].F := 1000; Lines1[82].CMD := 2; Lines1[82].Param := 0; // G1 Continuous [Op67 P1]
    Lines1[83].X := 253.042; Lines1[83].Z := 348.589; Lines1[83].F := 1000; Lines1[83].CMD := 2; Lines1[83].Param := 0; // G1 Continuous [Op67 P1]
    Lines1[84].X := 252.208; Lines1[84].Z := 350.136; Lines1[84].F := 1000; Lines1[84].CMD := 2; Lines1[84].Param := 0; // G1 Continuous [Op67 P1]
    Lines1[85].X := 251.358; Lines1[85].Z := 351.676; Lines1[85].F := 1000; Lines1[85].CMD := 2; Lines1[85].Param := 0; // G1 Continuous [Op67 P1]
    Lines1[86].X := 250.493; Lines1[86].Z := 353.206; Lines1[86].F := 1000; Lines1[86].CMD := 2; Lines1[86].Param := 0; // G1 Continuous [Op67 P1]
    Lines1[87].X := 249.486; Lines1[87].Z := 354.945; Lines1[87].F := 1000; Lines1[87].CMD := 2; Lines1[87].Param := 0; // G1 Continuous [Op67 P1]
    Lines1[88].X := 248.589; Lines1[88].Z := 356.457; Lines1[88].F := 1000; Lines1[88].CMD := 2; Lines1[88].Param := 0; // G1 Continuous [Op67 P1]
    Lines1[89].X := 247.547; Lines1[89].Z := 358.175; Lines1[89].F := 1000; Lines1[89].CMD := 2; Lines1[89].Param := 0; // G1 Continuous [Op67 P1]
    Lines1[90].X := 246.621; Lines1[90].Z := 359.669; Lines1[90].F := 1000; Lines1[90].CMD := 2; Lines1[90].Param := 0; // G1 Continuous [Op67 P1]
    Lines1[91].X := 245.546; Lines1[91].Z := 361.365; Lines1[91].F := 1000; Lines1[91].CMD := 2; Lines1[91].Param := 0; // G1 Continuous [Op67 P1]
    Lines1[92].X := 244.591; Lines1[92].Z := 362.841; Lines1[92].F := 1000; Lines1[92].CMD := 2; Lines1[92].Param := 0; // G1 Continuous [Op67 P1]
    Lines1[93].X := 243.484; Lines1[93].Z := 364.517; Lines1[93].F := 1000; Lines1[93].CMD := 2; Lines1[93].Param := 0; // G1 Continuous [Op67 P1]
    Lines1[94].X := 242.362; Lines1[94].Z := 366.182; Lines1[94].F := 1000; Lines1[94].CMD := 2; Lines1[94].Param := 0; // G1 Continuous [Op67 P1]
    Lines1[95].X := 241.224; Lines1[95].Z := 367.836; Lines1[95].F := 1000; Lines1[95].CMD := 2; Lines1[95].Param := 0; // G1 Continuous [Op67 P1]
    Lines1[96].X := 239.050; Lines1[96].Z := 370.908; Lines1[96].F := 1000; Lines1[96].CMD := 2; Lines1[96].Param := 0; // G1 Continuous [Op67 P1]
    Lines1[97].X := 237.870; Lines1[97].Z := 372.531; Lines1[97].F := 1000; Lines1[97].CMD := 2; Lines1[97].Param := 0; // G1 Continuous [Op67 P1]
    Lines1[98].X := 236.677; Lines1[98].Z := 374.142; Lines1[98].F := 1000; Lines1[98].CMD := 2; Lines1[98].Param := 0; // G1 Continuous [Op67 P1]
    Lines1[99].X := 236.677; Lines1[99].Z := 374.142; Lines1[99].F := 0; Lines1[99].CMD := 41; Lines1[99].Param := 2; // M41 (Clamp On) P2 [Op68 P1]

    // --- Lines2 (global lines 100..199) ---
    Lines2[0].X := 231.757; Lines2[0].Z := 372.999; Lines2[0].F := 0; Lines2[0].CMD := 0; Lines2[0].Param := 0; // G0 Rapid [Op68 P1]
    Lines2[1].X := 233.260; Lines2[1].Z := 371.671; Lines2[1].F := 1000; Lines2[1].CMD := 2; Lines2[1].Param := 0; // G1 Continuous [Op68 P1]
    Lines2[2].X := 234.565; Lines2[2].Z := 370.495; Lines2[2].F := 1000; Lines2[2].CMD := 2; Lines2[2].Param := 0; // G1 Continuous [Op68 P1]
    Lines2[3].X := 236.043; Lines2[3].Z := 369.134; Lines2[3].F := 1000; Lines2[3].CMD := 2; Lines2[3].Param := 0; // G1 Continuous [Op68 P1]
    Lines2[4].X := 237.324; Lines2[4].Z := 367.928; Lines2[4].F := 1000; Lines2[4].CMD := 2; Lines2[4].Param := 0; // G1 Continuous [Op68 P1]
    Lines2[5].X := 238.592; Lines2[5].Z := 366.708; Lines2[5].F := 1000; Lines2[5].CMD := 2; Lines2[5].Param := 0; // G1 Continuous [Op68 P1]
    Lines2[6].X := 239.846; Lines2[6].Z := 365.473; Lines2[6].F := 1000; Lines2[6].CMD := 2; Lines2[6].Param := 0; // G1 Continuous [Op68 P1]
    Lines2[7].X := 241.084; Lines2[7].Z := 364.222; Lines2[7].F := 1000; Lines2[7].CMD := 2; Lines2[7].Param := 0; // G1 Continuous [Op68 P1]
    Lines2[8].X := 242.131; Lines2[8].Z := 363.138; Lines2[8].F := 1000; Lines2[8].CMD := 2; Lines2[8].Param := 0; // G1 Continuous [Op68 P1]
    Lines2[9].X := 243.336; Lines2[9].Z := 361.859; Lines2[9].F := 1000; Lines2[9].CMD := 2; Lines2[9].Param := 0; // G1 Continuous [Op68 P1]
    Lines2[10].X := 244.354; Lines2[10].Z := 360.749; Lines2[10].F := 1000; Lines2[10].CMD := 2; Lines2[10].Param := 0; // G1 Continuous [Op68 P1]
    Lines2[11].X := 245.522; Lines2[11].Z := 359.439; Lines2[11].F := 1000; Lines2[11].CMD := 2; Lines2[11].Param := 0; // G1 Continuous [Op68 P1]
    Lines2[12].X := 246.506; Lines2[12].Z := 358.303; Lines2[12].F := 1000; Lines2[12].CMD := 2; Lines2[12].Param := 0; // G1 Continuous [Op68 P1]
    Lines2[13].X := 247.474; Lines2[13].Z := 357.155; Lines2[13].F := 1000; Lines2[13].CMD := 2; Lines2[13].Param := 0; // G1 Continuous [Op68 P1]
    Lines2[14].X := 248.423; Lines2[14].Z := 355.993; Lines2[14].F := 1000; Lines2[14].CMD := 2; Lines2[14].Param := 0; // G1 Continuous [Op68 P1]
    Lines2[15].X := 249.355; Lines2[15].Z := 354.819; Lines2[15].F := 1000; Lines2[15].CMD := 2; Lines2[15].Param := 0; // G1 Continuous [Op68 P1]
    Lines2[16].X := 250.267; Lines2[16].Z := 353.632; Lines2[16].F := 1000; Lines2[16].CMD := 2; Lines2[16].Param := 0; // G1 Continuous [Op68 P1]
    Lines2[17].X := 251.159; Lines2[17].Z := 352.431; Lines2[17].F := 1000; Lines2[17].CMD := 2; Lines2[17].Param := 0; // G1 Continuous [Op68 P1]
    Lines2[18].X := 252.032; Lines2[18].Z := 351.217; Lines2[18].F := 1000; Lines2[18].CMD := 2; Lines2[18].Param := 0; // G1 Continuous [Op68 P1]
    Lines2[19].X := 252.885; Lines2[19].Z := 349.991; Lines2[19].F := 1000; Lines2[19].CMD := 2; Lines2[19].Param := 0; // G1 Continuous [Op68 P1]
    Lines2[20].X := 253.719; Lines2[20].Z := 348.751; Lines2[20].F := 1000; Lines2[20].CMD := 2; Lines2[20].Param := 0; // G1 Continuous [Op68 P1]
    Lines2[21].X := 254.534; Lines2[21].Z := 347.499; Lines2[21].F := 1000; Lines2[21].CMD := 2; Lines2[21].Param := 0; // G1 Continuous [Op68 P1]
    Lines2[22].X := 255.329; Lines2[22].Z := 346.235; Lines2[22].F := 1000; Lines2[22].CMD := 2; Lines2[22].Param := 0; // G1 Continuous [Op68 P1]
    Lines2[23].X := 256.105; Lines2[23].Z := 344.959; Lines2[23].F := 1000; Lines2[23].CMD := 2; Lines2[23].Param := 0; // G1 Continuous [Op68 P1]
    Lines2[24].X := 256.987; Lines2[24].Z := 343.456; Lines2[24].F := 1000; Lines2[24].CMD := 2; Lines2[24].Param := 0; // G1 Continuous [Op68 P1]
    Lines2[25].X := 257.722; Lines2[25].Z := 342.154; Lines2[25].F := 1000; Lines2[25].CMD := 2; Lines2[25].Param := 0; // G1 Continuous [Op68 P1]
    Lines2[26].X := 258.439; Lines2[26].Z := 340.841; Lines2[26].F := 1000; Lines2[26].CMD := 2; Lines2[26].Param := 0; // G1 Continuous [Op68 P1]
    Lines2[27].X := 259.137; Lines2[27].Z := 339.517; Lines2[27].F := 1000; Lines2[27].CMD := 2; Lines2[27].Param := 0; // G1 Continuous [Op68 P1]
    Lines2[28].X := 259.928; Lines2[28].Z := 337.959; Lines2[28].F := 1000; Lines2[28].CMD := 2; Lines2[28].Param := 0; // G1 Continuous [Op68 P1]
    Lines2[29].X := 260.586; Lines2[29].Z := 336.611; Lines2[29].F := 1000; Lines2[29].CMD := 2; Lines2[29].Param := 0; // G1 Continuous [Op68 P1]
    Lines2[30].X := 261.330; Lines2[30].Z := 335.026; Lines2[30].F := 1000; Lines2[30].CMD := 2; Lines2[30].Param := 0; // G1 Continuous [Op68 P1]
    Lines2[31].X := 261.949; Lines2[31].Z := 333.656; Lines2[31].F := 1000; Lines2[31].CMD := 2; Lines2[31].Param := 0; // G1 Continuous [Op68 P1]
    Lines2[32].X := 262.648; Lines2[32].Z := 332.044; Lines2[32].F := 1000; Lines2[32].CMD := 2; Lines2[32].Param := 0; // G1 Continuous [Op68 P1]
    Lines2[33].X := 263.227; Lines2[33].Z := 330.653; Lines2[33].F := 1000; Lines2[33].CMD := 2; Lines2[33].Param := 0; // G1 Continuous [Op68 P1]
    Lines2[34].X := 263.881; Lines2[34].Z := 329.017; Lines2[34].F := 1000; Lines2[34].CMD := 2; Lines2[34].Param := 0; // G1 Continuous [Op68 P1]
    Lines2[35].X := 264.422; Lines2[35].Z := 327.605; Lines2[35].F := 1000; Lines2[35].CMD := 2; Lines2[35].Param := 0; // G1 Continuous [Op68 P1]
    Lines2[36].X := 265.031; Lines2[36].Z := 325.945; Lines2[36].F := 1000; Lines2[36].CMD := 2; Lines2[36].Param := 0; // G1 Continuous [Op68 P1]
    Lines2[37].X := 265.534; Lines2[37].Z := 324.513; Lines2[37].F := 1000; Lines2[37].CMD := 2; Lines2[37].Param := 0; // G1 Continuous [Op68 P1]
    Lines2[38].X := 266.100; Lines2[38].Z := 322.832; Lines2[38].F := 1000; Lines2[38].CMD := 2; Lines2[38].Param := 0; // G1 Continuous [Op68 P1]
    Lines2[39].X := 266.642; Lines2[39].Z := 321.139; Lines2[39].F := 1000; Lines2[39].CMD := 2; Lines2[39].Param := 0; // G1 Continuous [Op68 P1]
    Lines2[40].X := 267.160; Lines2[40].Z := 319.434; Lines2[40].F := 1000; Lines2[40].CMD := 2; Lines2[40].Param := 0; // G1 Continuous [Op68 P1]
    Lines2[41].X := 267.586; Lines2[41].Z := 317.964; Lines2[41].F := 1000; Lines2[41].CMD := 2; Lines2[41].Param := 0; // G1 Continuous [Op68 P1]
    Lines2[42].X := 268.062; Lines2[42].Z := 316.240; Lines2[42].F := 1000; Lines2[42].CMD := 2; Lines2[42].Param := 0; // G1 Continuous [Op68 P1]
    Lines2[43].X := 268.515; Lines2[43].Z := 314.505; Lines2[43].F := 1000; Lines2[43].CMD := 2; Lines2[43].Param := 0; // G1 Continuous [Op68 P1]
    Lines2[44].X := 268.946; Lines2[44].Z := 312.760; Lines2[44].F := 1000; Lines2[44].CMD := 2; Lines2[44].Param := 0; // G1 Continuous [Op68 P1]
    Lines2[45].X := 269.354; Lines2[45].Z := 311.006; Lines2[45].F := 1000; Lines2[45].CMD := 2; Lines2[45].Param := 0; // G1 Continuous [Op68 P1]
    Lines2[46].X := 269.740; Lines2[46].Z := 309.242; Lines2[46].F := 1000; Lines2[46].CMD := 2; Lines2[46].Param := 0; // G1 Continuous [Op68 P1]
    Lines2[47].X := 270.104; Lines2[47].Z := 307.470; Lines2[47].F := 1000; Lines2[47].CMD := 2; Lines2[47].Param := 0; // G1 Continuous [Op68 P1]
    Lines2[48].X := 270.447; Lines2[48].Z := 305.688; Lines2[48].F := 1000; Lines2[48].CMD := 2; Lines2[48].Param := 0; // G1 Continuous [Op68 P1]
    Lines2[49].X := 270.767; Lines2[49].Z := 303.898; Lines2[49].F := 1000; Lines2[49].CMD := 2; Lines2[49].Param := 0; // G1 Continuous [Op68 P1]
    Lines2[50].X := 271.066; Lines2[50].Z := 302.101; Lines2[50].F := 1000; Lines2[50].CMD := 2; Lines2[50].Param := 0; // G1 Continuous [Op68 P1]
    Lines2[51].X := 271.344; Lines2[51].Z := 300.295; Lines2[51].F := 1000; Lines2[51].CMD := 2; Lines2[51].Param := 0; // G1 Continuous [Op68 P1]
    Lines2[52].X := 271.600; Lines2[52].Z := 298.482; Lines2[52].F := 1000; Lines2[52].CMD := 2; Lines2[52].Param := 0; // G1 Continuous [Op68 P1]
    Lines2[53].X := 271.836; Lines2[53].Z := 296.662; Lines2[53].F := 1000; Lines2[53].CMD := 2; Lines2[53].Param := 0; // G1 Continuous [Op68 P1]
    Lines2[54].X := 272.050; Lines2[54].Z := 294.836; Lines2[54].F := 1000; Lines2[54].CMD := 2; Lines2[54].Param := 0; // G1 Continuous [Op68 P1]
    Lines2[55].X := 272.244; Lines2[55].Z := 293.003; Lines2[55].F := 1000; Lines2[55].CMD := 2; Lines2[55].Param := 0; // G1 Continuous [Op68 P1]
    Lines2[56].X := 272.418; Lines2[56].Z := 291.164; Lines2[56].F := 1000; Lines2[56].CMD := 2; Lines2[56].Param := 0; // G1 Continuous [Op68 P1]
    Lines2[57].X := 272.571; Lines2[57].Z := 289.319; Lines2[57].F := 1000; Lines2[57].CMD := 2; Lines2[57].Param := 0; // G1 Continuous [Op68 P1]
    Lines2[58].X := 272.704; Lines2[58].Z := 287.469; Lines2[58].F := 1000; Lines2[58].CMD := 2; Lines2[58].Param := 0; // G1 Continuous [Op68 P1]
    Lines2[59].X := 272.817; Lines2[59].Z := 285.614; Lines2[59].F := 1000; Lines2[59].CMD := 2; Lines2[59].Param := 0; // G1 Continuous [Op68 P1]
    Lines2[60].X := 272.923; Lines2[60].Z := 283.488; Lines2[60].F := 1000; Lines2[60].CMD := 2; Lines2[60].Param := 0; // G1 Continuous [Op68 P1]
    Lines2[61].X := 272.994; Lines2[61].Z := 281.623; Lines2[61].F := 1000; Lines2[61].CMD := 2; Lines2[61].Param := 0; // G1 Continuous [Op68 P1]
    Lines2[62].X := 273.045; Lines2[62].Z := 279.754; Lines2[62].F := 1000; Lines2[62].CMD := 2; Lines2[62].Param := 0; // G1 Continuous [Op68 P1]
    Lines2[63].X := 273.078; Lines2[63].Z := 277.882; Lines2[63].F := 1000; Lines2[63].CMD := 2; Lines2[63].Param := 0; // G1 Continuous [Op68 P1]
    Lines2[64].X := 273.091; Lines2[64].Z := 275.737; Lines2[64].F := 1000; Lines2[64].CMD := 2; Lines2[64].Param := 0; // G1 Continuous [Op68 P1]
    Lines2[65].X := 273.074; Lines2[65].Z := 273.051; Lines2[65].F := 1000; Lines2[65].CMD := 2; Lines2[65].Param := 0; // G1 Continuous [Op68 P1]
    Lines2[66].X := 273.011; Lines2[66].Z := 270.091; Lines2[66].F := 1000; Lines2[66].CMD := 2; Lines2[66].Param := 0; // G1 Continuous [Op68 P1]
    Lines2[67].X := 272.903; Lines2[67].Z := 267.126; Lines2[67].F := 1000; Lines2[67].CMD := 2; Lines2[67].Param := 0; // G1 Continuous [Op68 P1]
    Lines2[68].X := 272.750; Lines2[68].Z := 264.156; Lines2[68].F := 1000; Lines2[68].CMD := 2; Lines2[68].Param := 0; // G1 Continuous [Op68 P1]
    Lines2[69].X := 272.553; Lines2[69].Z := 261.185; Lines2[69].F := 1000; Lines2[69].CMD := 2; Lines2[69].Param := 0; // G1 Continuous [Op68 P1]
    Lines2[70].X := 272.313; Lines2[70].Z := 258.212; Lines2[70].F := 1000; Lines2[70].CMD := 2; Lines2[70].Param := 0; // G1 Continuous [Op68 P1]
    Lines2[71].X := 272.031; Lines2[71].Z := 255.239; Lines2[71].F := 1000; Lines2[71].CMD := 2; Lines2[71].Param := 0; // G1 Continuous [Op68 P1]
    Lines2[72].X := 271.707; Lines2[72].Z := 252.268; Lines2[72].F := 1000; Lines2[72].CMD := 2; Lines2[72].Param := 0; // G1 Continuous [Op68 P1]
    Lines2[73].X := 271.341; Lines2[73].Z := 249.299; Lines2[73].F := 1000; Lines2[73].CMD := 2; Lines2[73].Param := 0; // G1 Continuous [Op68 P1]
    Lines2[74].X := 270.935; Lines2[74].Z := 246.334; Lines2[74].F := 1000; Lines2[74].CMD := 2; Lines2[74].Param := 0; // G1 Continuous [Op68 P1]
    Lines2[75].X := 270.489; Lines2[75].Z := 243.375; Lines2[75].F := 1000; Lines2[75].CMD := 2; Lines2[75].Param := 0; // G1 Continuous [Op68 P1]
    Lines2[76].X := 269.958; Lines2[76].Z := 240.153; Lines2[76].F := 1000; Lines2[76].CMD := 2; Lines2[76].Param := 0; // G1 Continuous [Op68 P1]
    Lines2[77].X := 269.431; Lines2[77].Z := 237.209; Lines2[77].F := 1000; Lines2[77].CMD := 2; Lines2[77].Param := 0; // G1 Continuous [Op68 P1]
    Lines2[78].X := 268.813; Lines2[78].Z := 234.007; Lines2[78].F := 1000; Lines2[78].CMD := 2; Lines2[78].Param := 0; // G1 Continuous [Op68 P1]
    Lines2[79].X := 268.208; Lines2[79].Z := 231.082; Lines2[79].F := 1000; Lines2[79].CMD := 2; Lines2[79].Param := 0; // G1 Continuous [Op68 P1]
    Lines2[80].X := 267.506; Lines2[80].Z := 227.906; Lines2[80].F := 1000; Lines2[80].CMD := 2; Lines2[80].Param := 0; // G1 Continuous [Op68 P1]
    Lines2[81].X := 266.826; Lines2[81].Z := 225.007; Lines2[81].F := 1000; Lines2[81].CMD := 2; Lines2[81].Param := 0; // G1 Continuous [Op68 P1]
    Lines2[82].X := 266.044; Lines2[82].Z := 221.862; Lines2[82].F := 1000; Lines2[82].CMD := 2; Lines2[82].Param := 0; // G1 Continuous [Op68 P1]
    Lines2[83].X := 265.221; Lines2[83].Z := 218.736; Lines2[83].F := 1000; Lines2[83].CMD := 2; Lines2[83].Param := 0; // G1 Continuous [Op68 P1]
    Lines2[84].X := 264.359; Lines2[84].Z := 215.630; Lines2[84].F := 1000; Lines2[84].CMD := 2; Lines2[84].Param := 0; // G1 Continuous [Op68 P1]
    Lines2[85].X := 263.534; Lines2[85].Z := 212.802; Lines2[85].F := 1000; Lines2[85].CMD := 2; Lines2[85].Param := 0; // G1 Continuous [Op68 P1]
    Lines2[86].X := 262.598; Lines2[86].Z := 209.740; Lines2[86].F := 1000; Lines2[86].CMD := 2; Lines2[86].Param := 0; // G1 Continuous [Op68 P1]
    Lines2[87].X := 261.624; Lines2[87].Z := 206.703; Lines2[87].F := 1000; Lines2[87].CMD := 2; Lines2[87].Param := 0; // G1 Continuous [Op68 P1]
    Lines2[88].X := 260.614; Lines2[88].Z := 203.693; Lines2[88].F := 1000; Lines2[88].CMD := 2; Lines2[88].Param := 0; // G1 Continuous [Op68 P1]
    Lines2[89].X := 259.657; Lines2[89].Z := 200.959; Lines2[89].F := 1000; Lines2[89].CMD := 2; Lines2[89].Param := 0; // G1 Continuous [Op68 P1]
    Lines2[90].X := 258.580; Lines2[90].Z := 198.005; Lines2[90].F := 1000; Lines2[90].CMD := 2; Lines2[90].Param := 0; // G1 Continuous [Op68 P1]
    Lines2[91].X := 257.469; Lines2[91].Z := 195.083; Lines2[91].F := 1000; Lines2[91].CMD := 2; Lines2[91].Param := 0; // G1 Continuous [Op68 P1]
    Lines2[92].X := 256.325; Lines2[92].Z := 192.194; Lines2[92].F := 1000; Lines2[92].CMD := 2; Lines2[92].Param := 0; // G1 Continuous [Op68 P1]
    Lines2[93].X := 255.149; Lines2[93].Z := 189.340; Lines2[93].F := 1000; Lines2[93].CMD := 2; Lines2[93].Param := 0; // G1 Continuous [Op68 P1]
    Lines2[94].X := 253.942; Lines2[94].Z := 186.523; Lines2[94].F := 1000; Lines2[94].CMD := 2; Lines2[94].Param := 0; // G1 Continuous [Op68 P1]
    Lines2[95].X := 252.705; Lines2[95].Z := 183.745; Lines2[95].F := 1000; Lines2[95].CMD := 2; Lines2[95].Param := 0; // G1 Continuous [Op68 P1]
    Lines2[96].X := 251.438; Lines2[96].Z := 181.006; Lines2[96].F := 293; Lines2[96].CMD := 2; Lines2[96].Param := 0; // G1 Continuous [Op68 P1]
    Lines2[97].X := 247.987; Lines2[97].Z := 181.006; Lines2[97].F := 293; Lines2[97].CMD := 1; Lines2[97].Param := 0; // G1 Linear [Op69 P1]
    Lines2[98].X := 249.489; Lines2[98].Z := 183.922; Lines2[98].F := 1000; Lines2[98].CMD := 2; Lines2[98].Param := 0; // G1 Continuous [Op69 P1]
    Lines2[99].X := 250.848; Lines2[99].Z := 186.671; Lines2[99].F := 1000; Lines2[99].CMD := 2; Lines2[99].Param := 0; // G1 Continuous [Op69 P1]

    // --- Lines3 (global lines 200..299) ---
    Lines3[0].X := 252.179; Lines3[0].Z := 189.471; Lines3[0].F := 1000; Lines3[0].CMD := 2; Lines3[0].Param := 0; // G1 Continuous [Op69 P1]
    Lines3[1].X := 253.482; Lines3[1].Z := 192.321; Lines3[1].F := 1000; Lines3[1].CMD := 2; Lines3[1].Param := 0; // G1 Continuous [Op69 P1]
    Lines3[2].X := 254.860; Lines3[2].Z := 195.462; Lines3[2].F := 1000; Lines3[2].CMD := 2; Lines3[2].Param := 0; // G1 Continuous [Op69 P1]
    Lines3[3].X := 256.098; Lines3[3].Z := 198.408; Lines3[3].F := 1000; Lines3[3].CMD := 2; Lines3[3].Param := 0; // G1 Continuous [Op69 P1]
    Lines3[4].X := 257.305; Lines3[4].Z := 201.396; Lines3[4].F := 1000; Lines3[4].CMD := 2; Lines3[4].Param := 0; // G1 Continuous [Op69 P1]
    Lines3[5].X := 258.477; Lines3[5].Z := 204.425; Lines3[5].F := 1000; Lines3[5].CMD := 2; Lines3[5].Param := 0; // G1 Continuous [Op69 P1]
    Lines3[6].X := 259.614; Lines3[6].Z := 207.491; Lines3[6].F := 1000; Lines3[6].CMD := 2; Lines3[6].Param := 0; // G1 Continuous [Op69 P1]
    Lines3[7].X := 260.714; Lines3[7].Z := 210.593; Lines3[7].F := 1000; Lines3[7].CMD := 2; Lines3[7].Param := 0; // G1 Continuous [Op69 P1]
    Lines3[8].X := 261.776; Lines3[8].Z := 213.727; Lines3[8].F := 1000; Lines3[8].CMD := 2; Lines3[8].Param := 0; // G1 Continuous [Op69 P1]
    Lines3[9].X := 262.800; Lines3[9].Z := 216.893; Lines3[9].F := 1000; Lines3[9].CMD := 2; Lines3[9].Param := 0; // G1 Continuous [Op69 P1]
    Lines3[10].X := 263.782; Lines3[10].Z := 220.087; Lines3[10].F := 1000; Lines3[10].CMD := 2; Lines3[10].Param := 0; // G1 Continuous [Op69 P1]
    Lines3[11].X := 264.723; Lines3[11].Z := 223.307; Lines3[11].F := 1000; Lines3[11].CMD := 2; Lines3[11].Param := 0; // G1 Continuous [Op69 P1]
    Lines3[12].X := 265.621; Lines3[12].Z := 226.550; Lines3[12].F := 1000; Lines3[12].CMD := 2; Lines3[12].Param := 0; // G1 Continuous [Op69 P1]
    Lines3[13].X := 266.475; Lines3[13].Z := 229.815; Lines3[13].F := 1000; Lines3[13].CMD := 2; Lines3[13].Param := 0; // G1 Continuous [Op69 P1]
    Lines3[14].X := 267.283; Lines3[14].Z := 233.099; Lines3[14].F := 1000; Lines3[14].CMD := 2; Lines3[14].Param := 0; // G1 Continuous [Op69 P1]
    Lines3[15].X := 267.982; Lines3[15].Z := 236.125; Lines3[15].F := 1000; Lines3[15].CMD := 2; Lines3[15].Param := 0; // G1 Continuous [Op69 P1]
    Lines3[16].X := 268.699; Lines3[16].Z := 239.439; Lines3[16].F := 1000; Lines3[16].CMD := 2; Lines3[16].Param := 0; // G1 Continuous [Op69 P1]
    Lines3[17].X := 269.313; Lines3[17].Z := 242.487; Lines3[17].F := 1000; Lines3[17].CMD := 2; Lines3[17].Param := 0; // G1 Continuous [Op69 P1]
    Lines3[18].X := 269.934; Lines3[18].Z := 245.823; Lines3[18].F := 1000; Lines3[18].CMD := 2; Lines3[18].Param := 0; // G1 Continuous [Op69 P1]
    Lines3[19].X := 270.458; Lines3[19].Z := 248.887; Lines3[19].F := 1000; Lines3[19].CMD := 2; Lines3[19].Param := 0; // G1 Continuous [Op69 P1]
    Lines3[20].X := 270.978; Lines3[20].Z := 252.235; Lines3[20].F := 1000; Lines3[20].CMD := 2; Lines3[20].Param := 0; // G1 Continuous [Op69 P1]
    Lines3[21].X := 271.408; Lines3[21].Z := 255.308; Lines3[21].F := 1000; Lines3[21].CMD := 2; Lines3[21].Param := 0; // G1 Continuous [Op69 P1]
    Lines3[22].X := 271.823; Lines3[22].Z := 258.660; Lines3[22].F := 1000; Lines3[22].CMD := 2; Lines3[22].Param := 0; // G1 Continuous [Op69 P1]
    Lines3[23].X := 272.153; Lines3[23].Z := 261.732; Lines3[23].F := 1000; Lines3[23].CMD := 2; Lines3[23].Param := 0; // G1 Continuous [Op69 P1]
    Lines3[24].X := 272.435; Lines3[24].Z := 264.801; Lines3[24].F := 1000; Lines3[24].CMD := 2; Lines3[24].Param := 0; // G1 Continuous [Op69 P1]
    Lines3[25].X := 272.667; Lines3[25].Z := 267.866; Lines3[25].F := 1000; Lines3[25].CMD := 2; Lines3[25].Param := 0; // G1 Continuous [Op69 P1]
    Lines3[26].X := 272.848; Lines3[26].Z := 270.924; Lines3[26].F := 1000; Lines3[26].CMD := 2; Lines3[26].Param := 0; // G1 Continuous [Op69 P1]
    Lines3[27].X := 272.978; Lines3[27].Z := 273.974; Lines3[27].F := 1000; Lines3[27].CMD := 2; Lines3[27].Param := 0; // G1 Continuous [Op69 P1]
    Lines3[28].X := 273.054; Lines3[28].Z := 277.014; Lines3[28].F := 1000; Lines3[28].CMD := 2; Lines3[28].Param := 0; // G1 Continuous [Op69 P1]
    Lines3[29].X := 273.078; Lines3[29].Z := 279.768; Lines3[29].F := 1000; Lines3[29].CMD := 2; Lines3[29].Param := 0; // G1 Continuous [Op69 P1]
    Lines3[30].X := 273.067; Lines3[30].Z := 281.688; Lines3[30].F := 1000; Lines3[30].CMD := 2; Lines3[30].Param := 0; // G1 Continuous [Op69 P1]
    Lines3[31].X := 273.040; Lines3[31].Z := 283.330; Lines3[31].F := 1000; Lines3[31].CMD := 2; Lines3[31].Param := 0; // G1 Continuous [Op69 P1]
    Lines3[32].X := 272.936; Lines3[32].Z := 286.599; Lines3[32].F := 1000; Lines3[32].CMD := 2; Lines3[32].Param := 0; // G1 Continuous [Op69 P1]
    Lines3[33].X := 272.844; Lines3[33].Z := 288.497; Lines3[33].F := 1000; Lines3[33].CMD := 2; Lines3[33].Param := 0; // G1 Continuous [Op69 P1]
    Lines3[34].X := 272.747; Lines3[34].Z := 290.118; Lines3[34].F := 1000; Lines3[34].CMD := 2; Lines3[34].Param := 0; // G1 Continuous [Op69 P1]
    Lines3[35].X := 272.633; Lines3[35].Z := 291.732; Lines3[35].F := 1000; Lines3[35].CMD := 2; Lines3[35].Param := 0; // G1 Continuous [Op69 P1]
    Lines3[36].X := 272.501; Lines3[36].Z := 293.341; Lines3[36].F := 1000; Lines3[36].CMD := 2; Lines3[36].Param := 0; // G1 Continuous [Op69 P1]
    Lines3[37].X := 272.351; Lines3[37].Z := 294.943; Lines3[37].F := 1000; Lines3[37].CMD := 2; Lines3[37].Param := 0; // G1 Continuous [Op69 P1]
    Lines3[38].X := 272.184; Lines3[38].Z := 296.538; Lines3[38].F := 1000; Lines3[38].CMD := 2; Lines3[38].Param := 0; // G1 Continuous [Op69 P1]
    Lines3[39].X := 271.998; Lines3[39].Z := 298.126; Lines3[39].F := 1000; Lines3[39].CMD := 2; Lines3[39].Param := 0; // G1 Continuous [Op69 P1]
    Lines3[40].X := 271.795; Lines3[40].Z := 299.707; Lines3[40].F := 1000; Lines3[40].CMD := 2; Lines3[40].Param := 0; // G1 Continuous [Op69 P1]
    Lines3[41].X := 271.573; Lines3[41].Z := 301.281; Lines3[41].F := 1000; Lines3[41].CMD := 2; Lines3[41].Param := 0; // G1 Continuous [Op69 P1]
    Lines3[42].X := 271.333; Lines3[42].Z := 302.846; Lines3[42].F := 1000; Lines3[42].CMD := 2; Lines3[42].Param := 0; // G1 Continuous [Op69 P1]
    Lines3[43].X := 271.075; Lines3[43].Z := 304.403; Lines3[43].F := 1000; Lines3[43].CMD := 2; Lines3[43].Param := 0; // G1 Continuous [Op69 P1]
    Lines3[44].X := 270.797; Lines3[44].Z := 305.952; Lines3[44].F := 1000; Lines3[44].CMD := 2; Lines3[44].Param := 0; // G1 Continuous [Op69 P1]
    Lines3[45].X := 270.501; Lines3[45].Z := 307.492; Lines3[45].F := 1000; Lines3[45].CMD := 2; Lines3[45].Param := 0; // G1 Continuous [Op69 P1]
    Lines3[46].X := 270.185; Lines3[46].Z := 309.023; Lines3[46].F := 1000; Lines3[46].CMD := 2; Lines3[46].Param := 0; // G1 Continuous [Op69 P1]
    Lines3[47].X := 269.851; Lines3[47].Z := 310.545; Lines3[47].F := 1000; Lines3[47].CMD := 2; Lines3[47].Param := 0; // G1 Continuous [Op69 P1]
    Lines3[48].X := 269.497; Lines3[48].Z := 312.057; Lines3[48].F := 1000; Lines3[48].CMD := 2; Lines3[48].Param := 0; // G1 Continuous [Op69 P1]
    Lines3[49].X := 269.123; Lines3[49].Z := 313.559; Lines3[49].F := 1000; Lines3[49].CMD := 2; Lines3[49].Param := 0; // G1 Continuous [Op69 P1]
    Lines3[50].X := 268.730; Lines3[50].Z := 315.050; Lines3[50].F := 1000; Lines3[50].CMD := 2; Lines3[50].Param := 0; // G1 Continuous [Op69 P1]
    Lines3[51].X := 268.317; Lines3[51].Z := 316.532; Lines3[51].F := 1000; Lines3[51].CMD := 2; Lines3[51].Param := 0; // G1 Continuous [Op69 P1]
    Lines3[52].X := 267.957; Lines3[52].Z := 317.758; Lines3[52].F := 1000; Lines3[52].CMD := 2; Lines3[52].Param := 0; // G1 Continuous [Op69 P1]
    Lines3[53].X := 267.507; Lines3[53].Z := 319.219; Lines3[53].F := 1000; Lines3[53].CMD := 2; Lines3[53].Param := 0; // G1 Continuous [Op69 P1]
    Lines3[54].X := 267.037; Lines3[54].Z := 320.668; Lines3[54].F := 1000; Lines3[54].CMD := 2; Lines3[54].Param := 0; // G1 Continuous [Op69 P1]
    Lines3[55].X := 266.546; Lines3[55].Z := 322.107; Lines3[55].F := 1000; Lines3[55].CMD := 2; Lines3[55].Param := 0; // G1 Continuous [Op69 P1]
    Lines3[56].X := 266.121; Lines3[56].Z := 323.296; Lines3[56].F := 1000; Lines3[56].CMD := 2; Lines3[56].Param := 0; // G1 Continuous [Op69 P1]
    Lines3[57].X := 265.592; Lines3[57].Z := 324.712; Lines3[57].F := 1000; Lines3[57].CMD := 2; Lines3[57].Param := 0; // G1 Continuous [Op69 P1]
    Lines3[58].X := 265.136; Lines3[58].Z := 325.882; Lines3[58].F := 1000; Lines3[58].CMD := 2; Lines3[58].Param := 0; // G1 Continuous [Op69 P1]
    Lines3[59].X := 264.568; Lines3[59].Z := 327.275; Lines3[59].F := 1000; Lines3[59].CMD := 2; Lines3[59].Param := 0; // G1 Continuous [Op69 P1]
    Lines3[60].X := 264.079; Lines3[60].Z := 328.426; Lines3[60].F := 1000; Lines3[60].CMD := 2; Lines3[60].Param := 0; // G1 Continuous [Op69 P1]
    Lines3[61].X := 263.473; Lines3[61].Z := 329.795; Lines3[61].F := 1000; Lines3[61].CMD := 2; Lines3[61].Param := 0; // G1 Continuous [Op69 P1]
    Lines3[62].X := 262.951; Lines3[62].Z := 330.925; Lines3[62].F := 1000; Lines3[62].CMD := 2; Lines3[62].Param := 0; // G1 Continuous [Op69 P1]
    Lines3[63].X := 262.305; Lines3[63].Z := 332.269; Lines3[63].F := 1000; Lines3[63].CMD := 2; Lines3[63].Param := 0; // G1 Continuous [Op69 P1]
    Lines3[64].X := 261.750; Lines3[64].Z := 333.378; Lines3[64].F := 1000; Lines3[64].CMD := 2; Lines3[64].Param := 0; // G1 Continuous [Op69 P1]
    Lines3[65].X := 261.063; Lines3[65].Z := 334.696; Lines3[65].F := 1000; Lines3[65].CMD := 2; Lines3[65].Param := 0; // G1 Continuous [Op69 P1]
    Lines3[66].X := 260.475; Lines3[66].Z := 335.783; Lines3[66].F := 1000; Lines3[66].CMD := 2; Lines3[66].Param := 0; // G1 Continuous [Op69 P1]
    Lines3[67].X := 259.748; Lines3[67].Z := 337.073; Lines3[67].F := 1000; Lines3[67].CMD := 2; Lines3[67].Param := 0; // G1 Continuous [Op69 P1]
    Lines3[68].X := 259.125; Lines3[68].Z := 338.137; Lines3[68].F := 1000; Lines3[68].CMD := 2; Lines3[68].Param := 0; // G1 Continuous [Op69 P1]
    Lines3[69].X := 258.356; Lines3[69].Z := 339.400; Lines3[69].F := 1000; Lines3[69].CMD := 2; Lines3[69].Param := 0; // G1 Continuous [Op69 P1]
    Lines3[70].X := 257.699; Lines3[70].Z := 340.440; Lines3[70].F := 1000; Lines3[70].CMD := 2; Lines3[70].Param := 0; // G1 Continuous [Op69 P1]
    Lines3[71].X := 256.889; Lines3[71].Z := 341.674; Lines3[71].F := 1000; Lines3[71].CMD := 2; Lines3[71].Param := 0; // G1 Continuous [Op69 P1]
    Lines3[72].X := 256.196; Lines3[72].Z := 342.690; Lines3[72].F := 1000; Lines3[72].CMD := 2; Lines3[72].Param := 0; // G1 Continuous [Op69 P1]
    Lines3[73].X := 255.344; Lines3[73].Z := 343.893; Lines3[73].F := 1000; Lines3[73].CMD := 2; Lines3[73].Param := 0; // G1 Continuous [Op69 P1]
    Lines3[74].X := 254.615; Lines3[74].Z := 344.884; Lines3[74].F := 1000; Lines3[74].CMD := 2; Lines3[74].Param := 0; // G1 Continuous [Op69 P1]
    Lines3[75].X := 253.871; Lines3[75].Z := 345.862; Lines3[75].F := 1000; Lines3[75].CMD := 2; Lines3[75].Param := 0; // G1 Continuous [Op69 P1]
    Lines3[76].X := 253.110; Lines3[76].Z := 346.829; Lines3[76].F := 1000; Lines3[76].CMD := 2; Lines3[76].Param := 0; // G1 Continuous [Op69 P1]
    Lines3[77].X := 252.333; Lines3[77].Z := 347.783; Lines3[77].F := 1000; Lines3[77].CMD := 2; Lines3[77].Param := 0; // G1 Continuous [Op69 P1]
    Lines3[78].X := 251.539; Lines3[78].Z := 348.725; Lines3[78].F := 1000; Lines3[78].CMD := 2; Lines3[78].Param := 0; // G1 Continuous [Op69 P1]
    Lines3[79].X := 250.728; Lines3[79].Z := 349.654; Lines3[79].F := 1000; Lines3[79].CMD := 2; Lines3[79].Param := 0; // G1 Continuous [Op69 P1]
    Lines3[80].X := 249.901; Lines3[80].Z := 350.571; Lines3[80].F := 1000; Lines3[80].CMD := 2; Lines3[80].Param := 0; // G1 Continuous [Op69 P1]
    Lines3[81].X := 249.057; Lines3[81].Z := 351.475; Lines3[81].F := 1000; Lines3[81].CMD := 2; Lines3[81].Param := 0; // G1 Continuous [Op69 P1]
    Lines3[82].X := 248.196; Lines3[82].Z := 352.366; Lines3[82].F := 1000; Lines3[82].CMD := 2; Lines3[82].Param := 0; // G1 Continuous [Op69 P1]
    Lines3[83].X := 247.317; Lines3[83].Z := 353.244; Lines3[83].F := 1000; Lines3[83].CMD := 2; Lines3[83].Param := 0; // G1 Continuous [Op69 P1]
    Lines3[84].X := 246.422; Lines3[84].Z := 354.109; Lines3[84].F := 1000; Lines3[84].CMD := 2; Lines3[84].Param := 0; // G1 Continuous [Op69 P1]
    Lines3[85].X := 245.510; Lines3[85].Z := 354.960; Lines3[85].F := 1000; Lines3[85].CMD := 2; Lines3[85].Param := 0; // G1 Continuous [Op69 P1]
    Lines3[86].X := 244.582; Lines3[86].Z := 355.798; Lines3[86].F := 1000; Lines3[86].CMD := 2; Lines3[86].Param := 0; // G1 Continuous [Op69 P1]
    Lines3[87].X := 243.641; Lines3[87].Z := 356.625; Lines3[87].F := 1000; Lines3[87].CMD := 2; Lines3[87].Param := 0; // G1 Continuous [Op69 P1]
    Lines3[88].X := 242.494; Lines3[88].Z := 357.601; Lines3[88].F := 1000; Lines3[88].CMD := 2; Lines3[88].Param := 0; // G1 Continuous [Op69 P1]
    Lines3[89].X := 240.355; Lines3[89].Z := 359.350; Lines3[89].F := 1000; Lines3[89].CMD := 2; Lines3[89].Param := 0; // G1 Continuous [Op69 P1]
    Lines3[90].X := 239.172; Lines3[90].Z := 360.284; Lines3[90].F := 1000; Lines3[90].CMD := 2; Lines3[90].Param := 0; // G1 Continuous [Op69 P1]
    Lines3[91].X := 237.783; Lines3[91].Z := 361.358; Lines3[91].F := 1000; Lines3[91].CMD := 1; Lines3[91].Param := 0; // G1 Linear [Op69 P1]
    Lines3[92].X := 248.196; Lines3[92].Z := 352.366; Lines3[92].F := 1000; Lines3[92].CMD := 2; Lines3[92].Param := 0; // G1 Continuous [Op69 P1]
    Lines3[93].X := 256.196; Lines3[93].Z := 342.690; Lines3[93].F := 1000; Lines3[93].CMD := 2; Lines3[93].Param := 0; // G1 Continuous [Op69 P1]
    Lines3[94].X := 262.951; Lines3[94].Z := 330.925; Lines3[94].F := 1000; Lines3[94].CMD := 2; Lines3[94].Param := 0; // G1 Continuous [Op69 P1]
    Lines3[95].X := 267.957; Lines3[95].Z := 317.758; Lines3[95].F := 1000; Lines3[95].CMD := 2; Lines3[95].Param := 0; // G1 Continuous [Op69 P1]
    Lines3[96].X := 270.797; Lines3[96].Z := 305.952; Lines3[96].F := 1000; Lines3[96].CMD := 2; Lines3[96].Param := 0; // G1 Continuous [Op69 P1]
    Lines3[97].X := 272.633; Lines3[97].Z := 291.732; Lines3[97].F := 1000; Lines3[97].CMD := 2; Lines3[97].Param := 0; // G1 Continuous [Op69 P1]
    Lines3[98].X := 273.078; Lines3[98].Z := 279.768; Lines3[98].F := 1000; Lines3[98].CMD := 2; Lines3[98].Param := 0; // G1 Continuous [Op69 P1]
    Lines3[99].X := 272.547; Lines3[99].Z := 266.195; Lines3[99].F := 1000; Lines3[99].CMD := 2; Lines3[99].Param := 0; // G1 Continuous [Op69 P1]

    // --- Lines4 (global lines 300..399) ---
    Lines4[0].X := 270.951; Lines4[0].Z := 252.049; Lines4[0].F := 1000; Lines4[0].CMD := 1; Lines4[0].Param := 0; // G1 Linear [Op69 P1]
    Lines4[1].X := 272.539; Lines4[1].Z := 266.377; Lines4[1].F := 1000; Lines4[1].CMD := 2; Lines4[1].Param := 0; // G1 Continuous [Op70 P1]
    Lines4[2].X := 273.073; Lines4[2].Z := 280.437; Lines4[2].F := 1000; Lines4[2].CMD := 2; Lines4[2].Param := 0; // G1 Continuous [Op70 P1]
    Lines4[3].X := 272.490; Lines4[3].Z := 294.241; Lines4[3].F := 1000; Lines4[3].CMD := 2; Lines4[3].Param := 0; // G1 Continuous [Op70 P1]
    Lines4[4].X := 270.795; Lines4[4].Z := 307.111; Lines4[4].F := 1000; Lines4[4].CMD := 2; Lines4[4].Param := 0; // G1 Continuous [Op70 P1]
    Lines4[5].X := 267.545; Lines4[5].Z := 320.677; Lines4[5].F := 1000; Lines4[5].CMD := 2; Lines4[5].Param := 0; // G1 Continuous [Op70 P1]
    Lines4[6].X := 262.848; Lines4[6].Z := 333.182; Lines4[6].F := 1000; Lines4[6].CMD := 2; Lines4[6].Param := 0; // G1 Continuous [Op70 P1]
    Lines4[7].X := 256.288; Lines4[7].Z := 345.117; Lines4[7].F := 1000; Lines4[7].CMD := 2; Lines4[7].Param := 0; // G1 Continuous [Op70 P1]
    Lines4[8].X := 248.071; Lines4[8].Z := 355.609; Lines4[8].F := 1000; Lines4[8].CMD := 2; Lines4[8].Param := 0; // G1 Continuous [Op70 P1]
    Lines4[9].X := 237.761; Lines4[9].Z := 365.088; Lines4[9].F := 1000; Lines4[9].CMD := 2; Lines4[9].Param := 0; // G1 Continuous [Op70 P1]
    Lines4[10].X := 249.195; Lines4[10].Z := 181.006; Lines4[10].F := 0; Lines4[10].CMD := 0; Lines4[10].Param := 0; // G0 Rapid [Op71 P1]
    Lines4[11].X := 250.642; Lines4[11].Z := 183.940; Lines4[11].F := 1000; Lines4[11].CMD := 2; Lines4[11].Param := 0; // G1 Continuous [Op71 P1]
    Lines4[12].X := 251.947; Lines4[12].Z := 186.695; Lines4[12].F := 1000; Lines4[12].CMD := 2; Lines4[12].Param := 0; // G1 Continuous [Op71 P1]
    Lines4[13].X := 253.223; Lines4[13].Z := 189.493; Lines4[13].F := 1000; Lines4[13].CMD := 2; Lines4[13].Param := 0; // G1 Continuous [Op71 P1]
    Lines4[14].X := 254.469; Lines4[14].Z := 192.332; Lines4[14].F := 1000; Lines4[14].CMD := 2; Lines4[14].Param := 0; // G1 Continuous [Op71 P1]
    Lines4[15].X := 255.783; Lines4[15].Z := 195.451; Lines4[15].F := 1000; Lines4[15].CMD := 2; Lines4[15].Param := 0; // G1 Continuous [Op71 P1]
    Lines4[16].X := 256.961; Lines4[16].Z := 198.369; Lines4[16].F := 1000; Lines4[16].CMD := 2; Lines4[16].Param := 0; // G1 Continuous [Op71 P1]
    Lines4[17].X := 258.107; Lines4[17].Z := 201.323; Lines4[17].F := 1000; Lines4[17].CMD := 2; Lines4[17].Param := 0; // G1 Continuous [Op71 P1]
    Lines4[18].X := 259.218; Lines4[18].Z := 204.310; Lines4[18].F := 1000; Lines4[18].CMD := 2; Lines4[18].Param := 0; // G1 Continuous [Op71 P1]
    Lines4[19].X := 260.381; Lines4[19].Z := 207.582; Lines4[19].F := 1000; Lines4[19].CMD := 2; Lines4[19].Param := 0; // G1 Continuous [Op71 P1]
    Lines4[20].X := 261.417; Lines4[20].Z := 210.633; Lines4[20].F := 1000; Lines4[20].CMD := 2; Lines4[20].Param := 0; // G1 Continuous [Op71 P1]
    Lines4[21].X := 262.416; Lines4[21].Z := 213.713; Lines4[21].F := 1000; Lines4[21].CMD := 2; Lines4[21].Param := 0; // G1 Continuous [Op71 P1]
    Lines4[22].X := 263.377; Lines4[22].Z := 216.818; Lines4[22].F := 1000; Lines4[22].CMD := 2; Lines4[22].Param := 0; // G1 Continuous [Op71 P1]
    Lines4[23].X := 264.298; Lines4[23].Z := 219.948; Lines4[23].F := 1000; Lines4[23].CMD := 2; Lines4[23].Param := 0; // G1 Continuous [Op71 P1]
    Lines4[24].X := 265.179; Lines4[24].Z := 223.100; Lines4[24].F := 1000; Lines4[24].CMD := 2; Lines4[24].Param := 0; // G1 Continuous [Op71 P1]
    Lines4[25].X := 266.018; Lines4[25].Z := 226.274; Lines4[25].F := 1000; Lines4[25].CMD := 2; Lines4[25].Param := 0; // G1 Continuous [Op71 P1]
    Lines4[26].X := 266.816; Lines4[26].Z := 229.466; Lines4[26].F := 1000; Lines4[26].CMD := 2; Lines4[26].Param := 0; // G1 Continuous [Op71 P1]
    Lines4[27].X := 267.570; Lines4[27].Z := 232.675; Lines4[27].F := 1000; Lines4[27].CMD := 2; Lines4[27].Param := 0; // G1 Continuous [Op71 P1]
    Lines4[28].X := 268.281; Lines4[28].Z := 235.900; Lines4[28].F := 1000; Lines4[28].CMD := 2; Lines4[28].Param := 0; // G1 Continuous [Op71 P1]
    Lines4[29].X := 268.946; Lines4[29].Z := 239.138; Lines4[29].F := 1000; Lines4[29].CMD := 2; Lines4[29].Param := 0; // G1 Continuous [Op71 P1]
    Lines4[30].X := 269.516; Lines4[30].Z := 242.117; Lines4[30].F := 1000; Lines4[30].CMD := 2; Lines4[30].Param := 0; // G1 Continuous [Op71 P1]
    Lines4[31].X := 270.092; Lines4[31].Z := 245.376; Lines4[31].F := 1000; Lines4[31].CMD := 2; Lines4[31].Param := 0; // G1 Continuous [Op71 P1]
    Lines4[32].X := 270.621; Lines4[32].Z := 248.644; Lines4[32].F := 1000; Lines4[32].CMD := 2; Lines4[32].Param := 0; // G1 Continuous [Op71 P1]
    Lines4[33].X := 271.101; Lines4[33].Z := 251.917; Lines4[33].F := 1000; Lines4[33].CMD := 2; Lines4[33].Param := 0; // G1 Continuous [Op71 P1]
    Lines4[34].X := 271.498; Lines4[34].Z := 254.923; Lines4[34].F := 1000; Lines4[34].CMD := 2; Lines4[34].Param := 0; // G1 Continuous [Op71 P1]
    Lines4[35].X := 271.881; Lines4[35].Z := 258.204; Lines4[35].F := 1000; Lines4[35].CMD := 2; Lines4[35].Param := 0; // G1 Continuous [Op71 P1]
    Lines4[36].X := 272.188; Lines4[36].Z := 261.213; Lines4[36].F := 1000; Lines4[36].CMD := 2; Lines4[36].Param := 0; // G1 Continuous [Op71 P1]
    Lines4[37].X := 272.472; Lines4[37].Z := 264.494; Lines4[37].F := 1000; Lines4[37].CMD := 2; Lines4[37].Param := 0; // G1 Continuous [Op71 P1]
    Lines4[38].X := 272.686; Lines4[38].Z := 267.501; Lines4[38].F := 1000; Lines4[38].CMD := 2; Lines4[38].Param := 0; // G1 Continuous [Op71 P1]
    Lines4[39].X := 272.867; Lines4[39].Z := 270.777; Lines4[39].F := 1000; Lines4[39].CMD := 2; Lines4[39].Param := 0; // G1 Continuous [Op71 P1]
    Lines4[40].X := 272.985; Lines4[40].Z := 273.774; Lines4[40].F := 1000; Lines4[40].CMD := 2; Lines4[40].Param := 0; // G1 Continuous [Op71 P1]
    Lines4[41].X := 273.055; Lines4[41].Z := 276.766; Lines4[41].F := 1000; Lines4[41].CMD := 2; Lines4[41].Param := 0; // G1 Continuous [Op71 P1]
    Lines4[42].X := 273.078; Lines4[42].Z := 279.750; Lines4[42].F := 1000; Lines4[42].CMD := 2; Lines4[42].Param := 0; // G1 Continuous [Op71 P1]
    Lines4[43].X := 273.042; Lines4[43].Z := 283.265; Lines4[43].F := 1000; Lines4[43].CMD := 2; Lines4[43].Param := 0; // G1 Continuous [Op71 P1]
    Lines4[44].X := 272.994; Lines4[44].Z := 285.151; Lines4[44].F := 1000; Lines4[44].CMD := 2; Lines4[44].Param := 0; // G1 Continuous [Op71 P1]
    Lines4[45].X := 272.937; Lines4[45].Z := 286.765; Lines4[45].F := 1000; Lines4[45].CMD := 2; Lines4[45].Param := 0; // G1 Continuous [Op71 P1]
    Lines4[46].X := 272.852; Lines4[46].Z := 288.642; Lines4[46].F := 1000; Lines4[46].CMD := 2; Lines4[46].Param := 0; // G1 Continuous [Op71 P1]
    Lines4[47].X := 272.762; Lines4[47].Z := 290.247; Lines4[47].F := 1000; Lines4[47].CMD := 2; Lines4[47].Param := 0; // G1 Continuous [Op71 P1]
    Lines4[48].X := 272.537; Lines4[48].Z := 293.445; Lines4[48].F := 1000; Lines4[48].CMD := 2; Lines4[48].Param := 0; // G1 Continuous [Op71 P1]
    Lines4[49].X := 272.377; Lines4[49].Z := 295.302; Lines4[49].F := 1000; Lines4[49].CMD := 2; Lines4[49].Param := 0; // G1 Continuous [Op71 P1]
    Lines4[50].X := 272.223; Lines4[50].Z := 296.888; Lines4[50].F := 1000; Lines4[50].CMD := 2; Lines4[50].Param := 0; // G1 Continuous [Op71 P1]
    Lines4[51].X := 271.868; Lines4[51].Z := 300.045; Lines4[51].F := 1000; Lines4[51].CMD := 2; Lines4[51].Param := 0; // G1 Continuous [Op71 P1]
    Lines4[52].X := 271.449; Lines4[52].Z := 303.180; Lines4[52].F := 1000; Lines4[52].CMD := 2; Lines4[52].Param := 0; // G1 Continuous [Op71 P1]
    Lines4[53].X := 270.965; Lines4[53].Z := 306.291; Lines4[53].F := 1000; Lines4[53].CMD := 2; Lines4[53].Param := 0; // G1 Continuous [Op71 P1]
    Lines4[54].X := 270.652; Lines4[54].Z := 308.094; Lines4[54].F := 1000; Lines4[54].CMD := 2; Lines4[54].Param := 0; // G1 Continuous [Op71 P1]
    Lines4[55].X := 270.366; Lines4[55].Z := 309.632; Lines4[55].F := 1000; Lines4[55].CMD := 2; Lines4[55].Param := 0; // G1 Continuous [Op71 P1]
    Lines4[56].X := 270.064; Lines4[56].Z := 311.163; Lines4[56].F := 1000; Lines4[56].CMD := 2; Lines4[56].Param := 0; // G1 Continuous [Op71 P1]
    Lines4[57].X := 269.744; Lines4[57].Z := 312.687; Lines4[57].F := 1000; Lines4[57].CMD := 2; Lines4[57].Param := 0; // G1 Continuous [Op71 P1]
    Lines4[58].X := 269.408; Lines4[58].Z := 314.203; Lines4[58].F := 1000; Lines4[58].CMD := 2; Lines4[58].Param := 0; // G1 Continuous [Op71 P1]
    Lines4[59].X := 269.055; Lines4[59].Z := 315.712; Lines4[59].F := 1000; Lines4[59].CMD := 2; Lines4[59].Param := 0; // G1 Continuous [Op71 P1]
    Lines4[60].X := 268.684; Lines4[60].Z := 317.213; Lines4[60].F := 1000; Lines4[60].CMD := 2; Lines4[60].Param := 0; // G1 Continuous [Op71 P1]
    Lines4[61].X := 268.296; Lines4[61].Z := 318.707; Lines4[61].F := 1000; Lines4[61].CMD := 2; Lines4[61].Param := 0; // G1 Continuous [Op71 P1]
    Lines4[62].X := 267.891; Lines4[62].Z := 320.191; Lines4[62].F := 1000; Lines4[62].CMD := 2; Lines4[62].Param := 0; // G1 Continuous [Op71 P1]
    Lines4[63].X := 267.468; Lines4[63].Z := 321.667; Lines4[63].F := 1000; Lines4[63].CMD := 2; Lines4[63].Param := 0; // G1 Continuous [Op71 P1]
    Lines4[64].X := 267.028; Lines4[64].Z := 323.135; Lines4[64].F := 1000; Lines4[64].CMD := 2; Lines4[64].Param := 0; // G1 Continuous [Op71 P1]
    Lines4[65].X := 266.570; Lines4[65].Z := 324.593; Lines4[65].F := 1000; Lines4[65].CMD := 2; Lines4[65].Param := 0; // G1 Continuous [Op71 P1]
    Lines4[66].X := 266.094; Lines4[66].Z := 326.043; Lines4[66].F := 1000; Lines4[66].CMD := 2; Lines4[66].Param := 0; // G1 Continuous [Op71 P1]
    Lines4[67].X := 265.600; Lines4[67].Z := 327.483; Lines4[67].F := 1000; Lines4[67].CMD := 2; Lines4[67].Param := 0; // G1 Continuous [Op71 P1]
    Lines4[68].X := 264.646; Lines4[68].Z := 330.097; Lines4[68].F := 1000; Lines4[68].CMD := 2; Lines4[68].Param := 0; // G1 Continuous [Op71 P1]
    Lines4[69].X := 264.101; Lines4[69].Z := 331.509; Lines4[69].F := 1000; Lines4[69].CMD := 2; Lines4[69].Param := 0; // G1 Continuous [Op71 P1]
    Lines4[70].X := 263.536; Lines4[70].Z := 332.910; Lines4[70].F := 1000; Lines4[70].CMD := 2; Lines4[70].Param := 0; // G1 Continuous [Op71 P1]
    Lines4[71].X := 262.953; Lines4[71].Z := 334.302; Lines4[71].F := 1000; Lines4[71].CMD := 2; Lines4[71].Param := 0; // G1 Continuous [Op71 P1]
    Lines4[72].X := 262.453; Lines4[72].Z := 335.453; Lines4[72].F := 1000; Lines4[72].CMD := 2; Lines4[72].Param := 0; // G1 Continuous [Op71 P1]
    Lines4[73].X := 261.836; Lines4[73].Z := 336.824; Lines4[73].F := 1000; Lines4[73].CMD := 2; Lines4[73].Param := 0; // G1 Continuous [Op71 P1]
    Lines4[74].X := 261.200; Lines4[74].Z := 338.184; Lines4[74].F := 1000; Lines4[74].CMD := 2; Lines4[74].Param := 0; // G1 Continuous [Op71 P1]
    Lines4[75].X := 260.545; Lines4[75].Z := 339.533; Lines4[75].F := 1000; Lines4[75].CMD := 2; Lines4[75].Param := 0; // G1 Continuous [Op71 P1]
    Lines4[76].X := 259.984; Lines4[76].Z := 340.648; Lines4[76].F := 1000; Lines4[76].CMD := 2; Lines4[76].Param := 0; // G1 Continuous [Op71 P1]
    Lines4[77].X := 259.294; Lines4[77].Z := 341.975; Lines4[77].F := 1000; Lines4[77].CMD := 2; Lines4[77].Param := 0; // G1 Continuous [Op71 P1]
    Lines4[78].X := 258.584; Lines4[78].Z := 343.290; Lines4[78].F := 1000; Lines4[78].CMD := 2; Lines4[78].Param := 0; // G1 Continuous [Op71 P1]
    Lines4[79].X := 257.855; Lines4[79].Z := 344.593; Lines4[79].F := 1000; Lines4[79].CMD := 2; Lines4[79].Param := 0; // G1 Continuous [Op71 P1]
    Lines4[80].X := 257.232; Lines4[80].Z := 345.669; Lines4[80].F := 1000; Lines4[80].CMD := 2; Lines4[80].Param := 0; // G1 Continuous [Op71 P1]
    Lines4[81].X := 256.466; Lines4[81].Z := 346.949; Lines4[81].F := 1000; Lines4[81].CMD := 2; Lines4[81].Param := 0; // G1 Continuous [Op71 P1]
    Lines4[82].X := 255.813; Lines4[82].Z := 348.006; Lines4[82].F := 1000; Lines4[82].CMD := 2; Lines4[82].Param := 0; // G1 Continuous [Op71 P1]
    Lines4[83].X := 255.011; Lines4[83].Z := 349.262; Lines4[83].F := 1000; Lines4[83].CMD := 2; Lines4[83].Param := 0; // G1 Continuous [Op71 P1]
    Lines4[84].X := 254.328; Lines4[84].Z := 350.298; Lines4[84].F := 1000; Lines4[84].CMD := 2; Lines4[84].Param := 0; // G1 Continuous [Op71 P1]
    Lines4[85].X := 253.489; Lines4[85].Z := 351.530; Lines4[85].F := 1000; Lines4[85].CMD := 2; Lines4[85].Param := 0; // G1 Continuous [Op71 P1]
    Lines4[86].X := 252.775; Lines4[86].Z := 352.545; Lines4[86].F := 1000; Lines4[86].CMD := 2; Lines4[86].Param := 0; // G1 Continuous [Op71 P1]
    Lines4[87].X := 251.899; Lines4[87].Z := 353.751; Lines4[87].F := 1000; Lines4[87].CMD := 2; Lines4[87].Param := 0; // G1 Continuous [Op71 P1]
    Lines4[88].X := 251.153; Lines4[88].Z := 354.746; Lines4[88].F := 1000; Lines4[88].CMD := 2; Lines4[88].Param := 0; // G1 Continuous [Op71 P1]
    Lines4[89].X := 250.239; Lines4[89].Z := 355.926; Lines4[89].F := 1000; Lines4[89].CMD := 2; Lines4[89].Param := 0; // G1 Continuous [Op71 P1]
    Lines4[90].X := 249.462; Lines4[90].Z := 356.898; Lines4[90].F := 1000; Lines4[90].CMD := 2; Lines4[90].Param := 0; // G1 Continuous [Op71 P1]
    Lines4[91].X := 248.671; Lines4[91].Z := 357.860; Lines4[91].F := 1000; Lines4[91].CMD := 2; Lines4[91].Param := 0; // G1 Continuous [Op71 P1]
    Lines4[92].X := 247.864; Lines4[92].Z := 358.812; Lines4[92].F := 1000; Lines4[92].CMD := 2; Lines4[92].Param := 0; // G1 Continuous [Op71 P1]
    Lines4[93].X := 247.044; Lines4[93].Z := 359.753; Lines4[93].F := 1000; Lines4[93].CMD := 2; Lines4[93].Param := 0; // G1 Continuous [Op71 P1]
    Lines4[94].X := 246.041; Lines4[94].Z := 360.869; Lines4[94].F := 1000; Lines4[94].CMD := 2; Lines4[94].Param := 0; // G1 Continuous [Op71 P1]
    Lines4[95].X := 245.191; Lines4[95].Z := 361.788; Lines4[95].F := 1000; Lines4[95].CMD := 2; Lines4[95].Param := 0; // G1 Continuous [Op71 P1]
    Lines4[96].X := 244.157; Lines4[96].Z := 362.879; Lines4[96].F := 1000; Lines4[96].CMD := 2; Lines4[96].Param := 0; // G1 Continuous [Op71 P1]
    Lines4[97].X := 242.048; Lines4[97].Z := 365.025; Lines4[97].F := 1000; Lines4[97].CMD := 2; Lines4[97].Param := 0; // G1 Continuous [Op71 P1]
    Lines4[98].X := 239.898; Lines4[98].Z := 367.126; Lines4[98].F := 1000; Lines4[98].CMD := 2; Lines4[98].Param := 0; // G1 Continuous [Op71 P1]
    Lines4[99].X := 239.390; Lines4[99].Z := 349.475; Lines4[99].F := 0; Lines4[99].CMD := 0; Lines4[99].Param := 0; // G0 Rapid [Op72 P1]

    // --- Lines5 (global lines 400..499) ---
    Lines5[0].X := 240.616; Lines5[0].Z := 349.205; Lines5[0].F := 1000; Lines5[0].CMD := 2; Lines5[0].Param := 0; // G1 Continuous [Op72 P1]
    Lines5[1].X := 241.588; Lines5[1].Z := 348.973; Lines5[1].F := 1000; Lines5[1].CMD := 2; Lines5[1].Param := 0; // G1 Continuous [Op72 P1]
    Lines5[2].X := 242.545; Lines5[2].Z := 348.723; Lines5[2].F := 1000; Lines5[2].CMD := 2; Lines5[2].Param := 0; // G1 Continuous [Op72 P1]
    Lines5[3].X := 243.484; Lines5[3].Z := 348.453; Lines5[3].F := 1000; Lines5[3].CMD := 2; Lines5[3].Param := 0; // G1 Continuous [Op72 P1]
    Lines5[4].X := 244.407; Lines5[4].Z := 348.164; Lines5[4].F := 1000; Lines5[4].CMD := 2; Lines5[4].Param := 0; // G1 Continuous [Op72 P1]
    Lines5[5].X := 245.312; Lines5[5].Z := 347.856; Lines5[5].F := 1000; Lines5[5].CMD := 2; Lines5[5].Param := 0; // G1 Continuous [Op72 P1]
    Lines5[6].X := 246.201; Lines5[6].Z := 347.529; Lines5[6].F := 1000; Lines5[6].CMD := 2; Lines5[6].Param := 0; // G1 Continuous [Op72 P1]
    Lines5[7].X := 247.289; Lines5[7].Z := 347.094; Lines5[7].F := 1000; Lines5[7].CMD := 2; Lines5[7].Param := 0; // G1 Continuous [Op72 P1]
    Lines5[8].X := 248.141; Lines5[8].Z := 346.725; Lines5[8].F := 1000; Lines5[8].CMD := 2; Lines5[8].Param := 0; // G1 Continuous [Op72 P1]
    Lines5[9].X := 248.977; Lines5[9].Z := 346.338; Lines5[9].F := 1000; Lines5[9].CMD := 2; Lines5[9].Param := 0; // G1 Continuous [Op72 P1]
    Lines5[10].X := 249.796; Lines5[10].Z := 345.933; Lines5[10].F := 1000; Lines5[10].CMD := 2; Lines5[10].Param := 0; // G1 Continuous [Op72 P1]
    Lines5[11].X := 250.797; Lines5[11].Z := 345.402; Lines5[11].F := 1000; Lines5[11].CMD := 2; Lines5[11].Param := 0; // G1 Continuous [Op72 P1]
    Lines5[12].X := 251.580; Lines5[12].Z := 344.957; Lines5[12].F := 1000; Lines5[12].CMD := 2; Lines5[12].Param := 0; // G1 Continuous [Op72 P1]
    Lines5[13].X := 252.347; Lines5[13].Z := 344.494; Lines5[13].F := 1000; Lines5[13].CMD := 2; Lines5[13].Param := 0; // G1 Continuous [Op72 P1]
    Lines5[14].X := 253.098; Lines5[14].Z := 344.014; Lines5[14].F := 1000; Lines5[14].CMD := 2; Lines5[14].Param := 0; // G1 Continuous [Op72 P1]
    Lines5[15].X := 254.015; Lines5[15].Z := 343.391; Lines5[15].F := 1000; Lines5[15].CMD := 2; Lines5[15].Param := 0; // G1 Continuous [Op72 P1]
    Lines5[16].X := 254.730; Lines5[16].Z := 342.873; Lines5[16].F := 1000; Lines5[16].CMD := 2; Lines5[16].Param := 0; // G1 Continuous [Op72 P1]
    Lines5[17].X := 255.431; Lines5[17].Z := 342.338; Lines5[17].F := 1000; Lines5[17].CMD := 2; Lines5[17].Param := 0; // G1 Continuous [Op72 P1]
    Lines5[18].X := 256.116; Lines5[18].Z := 341.787; Lines5[18].F := 1000; Lines5[18].CMD := 2; Lines5[18].Param := 0; // G1 Continuous [Op72 P1]
    Lines5[19].X := 256.950; Lines5[19].Z := 341.075; Lines5[19].F := 1000; Lines5[19].CMD := 2; Lines5[19].Param := 0; // G1 Continuous [Op72 P1]
    Lines5[20].X := 257.601; Lines5[20].Z := 340.488; Lines5[20].F := 1000; Lines5[20].CMD := 2; Lines5[20].Param := 0; // G1 Continuous [Op72 P1]
    Lines5[21].X := 258.393; Lines5[21].Z := 339.731; Lines5[21].F := 1000; Lines5[21].CMD := 2; Lines5[21].Param := 0; // G1 Continuous [Op72 P1]
    Lines5[22].X := 259.009; Lines5[22].Z := 339.109; Lines5[22].F := 1000; Lines5[22].CMD := 2; Lines5[22].Param := 0; // G1 Continuous [Op72 P1]
    Lines5[23].X := 259.760; Lines5[23].Z := 338.308; Lines5[23].F := 1000; Lines5[23].CMD := 2; Lines5[23].Param := 0; // G1 Continuous [Op72 P1]
    Lines5[24].X := 260.343; Lines5[24].Z := 337.651; Lines5[24].F := 1000; Lines5[24].CMD := 2; Lines5[24].Param := 0; // G1 Continuous [Op72 P1]
    Lines5[25].X := 261.052; Lines5[25].Z := 336.808; Lines5[25].F := 1000; Lines5[25].CMD := 2; Lines5[25].Param := 0; // G1 Continuous [Op72 P1]
    Lines5[26].X := 261.603; Lines5[26].Z := 336.118; Lines5[26].F := 1000; Lines5[26].CMD := 2; Lines5[26].Param := 0; // G1 Continuous [Op72 P1]
    Lines5[27].X := 262.271; Lines5[27].Z := 335.234; Lines5[27].F := 1000; Lines5[27].CMD := 2; Lines5[27].Param := 0; // G1 Continuous [Op72 P1]
    Lines5[28].X := 262.789; Lines5[28].Z := 334.510; Lines5[28].F := 1000; Lines5[28].CMD := 2; Lines5[28].Param := 0; // G1 Continuous [Op72 P1]
    Lines5[29].X := 263.417; Lines5[29].Z := 333.586; Lines5[29].F := 1000; Lines5[29].CMD := 2; Lines5[29].Param := 0; // G1 Continuous [Op72 P1]
    Lines5[30].X := 263.904; Lines5[30].Z := 332.832; Lines5[30].F := 1000; Lines5[30].CMD := 2; Lines5[30].Param := 0; // G1 Continuous [Op72 P1]
    Lines5[31].X := 264.493; Lines5[31].Z := 331.869; Lines5[31].F := 1000; Lines5[31].CMD := 2; Lines5[31].Param := 0; // G1 Continuous [Op72 P1]
    Lines5[32].X := 264.949; Lines5[32].Z := 331.083; Lines5[32].F := 1000; Lines5[32].CMD := 2; Lines5[32].Param := 0; // G1 Continuous [Op72 P1]
    Lines5[33].X := 265.499; Lines5[33].Z := 330.082; Lines5[33].F := 1000; Lines5[33].CMD := 2; Lines5[33].Param := 0; // G1 Continuous [Op72 P1]
    Lines5[34].X := 265.924; Lines5[34].Z := 329.267; Lines5[34].F := 1000; Lines5[34].CMD := 2; Lines5[34].Param := 0; // G1 Continuous [Op72 P1]
    Lines5[35].X := 266.436; Lines5[35].Z := 328.230; Lines5[35].F := 1000; Lines5[35].CMD := 2; Lines5[35].Param := 0; // G1 Continuous [Op72 P1]
    Lines5[36].X := 266.830; Lines5[36].Z := 327.386; Lines5[36].F := 1000; Lines5[36].CMD := 2; Lines5[36].Param := 0; // G1 Continuous [Op72 P1]
    Lines5[37].X := 267.305; Lines5[37].Z := 326.314; Lines5[37].F := 1000; Lines5[37].CMD := 2; Lines5[37].Param := 0; // G1 Continuous [Op72 P1]
    Lines5[38].X := 267.759; Lines5[38].Z := 325.222; Lines5[38].F := 1000; Lines5[38].CMD := 2; Lines5[38].Param := 0; // G1 Continuous [Op72 P1]
    Lines5[39].X := 268.193; Lines5[39].Z := 324.112; Lines5[39].F := 1000; Lines5[39].CMD := 2; Lines5[39].Param := 0; // G1 Continuous [Op72 P1]
    Lines5[40].X := 268.526; Lines5[40].Z := 323.211; Lines5[40].F := 1000; Lines5[40].CMD := 2; Lines5[40].Param := 0; // G1 Continuous [Op72 P1]
    Lines5[41].X := 268.924; Lines5[41].Z := 322.067; Lines5[41].F := 1000; Lines5[41].CMD := 2; Lines5[41].Param := 0; // G1 Continuous [Op72 P1]
    Lines5[42].X := 269.302; Lines5[42].Z := 320.907; Lines5[42].F := 1000; Lines5[42].CMD := 2; Lines5[42].Param := 0; // G1 Continuous [Op72 P1]
    Lines5[43].X := 269.660; Lines5[43].Z := 319.729; Lines5[43].F := 1000; Lines5[43].CMD := 2; Lines5[43].Param := 0; // G1 Continuous [Op72 P1]
    Lines5[44].X := 270.000; Lines5[44].Z := 318.534; Lines5[44].F := 1000; Lines5[44].CMD := 2; Lines5[44].Param := 0; // G1 Continuous [Op72 P1]
    Lines5[45].X := 270.320; Lines5[45].Z := 317.322; Lines5[45].F := 1000; Lines5[45].CMD := 2; Lines5[45].Param := 0; // G1 Continuous [Op72 P1]
    Lines5[46].X := 270.621; Lines5[46].Z := 316.094; Lines5[46].F := 1000; Lines5[46].CMD := 2; Lines5[46].Param := 0; // G1 Continuous [Op72 P1]
    Lines5[47].X := 270.903; Lines5[47].Z := 314.850; Lines5[47].F := 1000; Lines5[47].CMD := 2; Lines5[47].Param := 0; // G1 Continuous [Op72 P1]
    Lines5[48].X := 271.167; Lines5[48].Z := 313.591; Lines5[48].F := 1000; Lines5[48].CMD := 2; Lines5[48].Param := 0; // G1 Continuous [Op72 P1]
    Lines5[49].X := 271.412; Lines5[49].Z := 312.317; Lines5[49].F := 1000; Lines5[49].CMD := 2; Lines5[49].Param := 0; // G1 Continuous [Op72 P1]
    Lines5[50].X := 271.640; Lines5[50].Z := 311.027; Lines5[50].F := 1000; Lines5[50].CMD := 2; Lines5[50].Param := 0; // G1 Continuous [Op72 P1]
    Lines5[51].X := 271.849; Lines5[51].Z := 309.724; Lines5[51].F := 1000; Lines5[51].CMD := 2; Lines5[51].Param := 0; // G1 Continuous [Op72 P1]
    Lines5[52].X := 272.041; Lines5[52].Z := 308.406; Lines5[52].F := 1000; Lines5[52].CMD := 2; Lines5[52].Param := 0; // G1 Continuous [Op72 P1]
    Lines5[53].X := 272.215; Lines5[53].Z := 307.075; Lines5[53].F := 1000; Lines5[53].CMD := 2; Lines5[53].Param := 0; // G1 Continuous [Op72 P1]
    Lines5[54].X := 272.372; Lines5[54].Z := 305.731; Lines5[54].F := 1000; Lines5[54].CMD := 2; Lines5[54].Param := 0; // G1 Continuous [Op72 P1]
    Lines5[55].X := 272.511; Lines5[55].Z := 304.373; Lines5[55].F := 1000; Lines5[55].CMD := 2; Lines5[55].Param := 0; // G1 Continuous [Op72 P1]
    Lines5[56].X := 272.634; Lines5[56].Z := 303.003; Lines5[56].F := 1000; Lines5[56].CMD := 2; Lines5[56].Param := 0; // G1 Continuous [Op72 P1]
    Lines5[57].X := 272.740; Lines5[57].Z := 301.621; Lines5[57].F := 1000; Lines5[57].CMD := 2; Lines5[57].Param := 0; // G1 Continuous [Op72 P1]
    Lines5[58].X := 272.902; Lines5[58].Z := 298.822; Lines5[58].F := 1000; Lines5[58].CMD := 2; Lines5[58].Param := 0; // G1 Continuous [Op72 P1]
    Lines5[59].X := 272.999; Lines5[59].Z := 295.978; Lines5[59].F := 1000; Lines5[59].CMD := 2; Lines5[59].Param := 0; // G1 Continuous [Op72 P1]
    Lines5[60].X := 273.024; Lines5[60].Z := 294.541; Lines5[60].F := 1000; Lines5[60].CMD := 2; Lines5[60].Param := 0; // G1 Continuous [Op72 P1]
    Lines5[61].X := 273.034; Lines5[61].Z := 292.802; Lines5[61].F := 1000; Lines5[61].CMD := 2; Lines5[61].Param := 0; // G1 Continuous [Op72 P1]
    Lines5[62].X := 273.001; Lines5[62].Z := 289.875; Lines5[62].F := 1000; Lines5[62].CMD := 2; Lines5[62].Param := 0; // G1 Continuous [Op72 P1]
    Lines5[63].X := 272.962; Lines5[63].Z := 288.398; Lines5[63].F := 1000; Lines5[63].CMD := 2; Lines5[63].Param := 0; // G1 Continuous [Op72 P1]
    Lines5[64].X := 272.896; Lines5[64].Z := 286.615; Lines5[64].F := 1000; Lines5[64].CMD := 2; Lines5[64].Param := 0; // G1 Continuous [Op72 P1]
    Lines5[65].X := 272.739; Lines5[65].Z := 283.617; Lines5[65].F := 1000; Lines5[65].CMD := 2; Lines5[65].Param := 0; // G1 Continuous [Op72 P1]
    Lines5[66].X := 272.502; Lines5[66].Z := 280.286; Lines5[66].F := 1000; Lines5[66].CMD := 2; Lines5[66].Param := 0; // G1 Continuous [Op72 P1]
    Lines5[67].X := 272.199; Lines5[67].Z := 276.924; Lines5[67].F := 1000; Lines5[67].CMD := 2; Lines5[67].Param := 0; // G1 Continuous [Op72 P1]
    Lines5[68].X := 271.831; Lines5[68].Z := 273.535; Lines5[68].F := 1000; Lines5[68].CMD := 2; Lines5[68].Param := 0; // G1 Continuous [Op72 P1]
    Lines5[69].X := 271.402; Lines5[69].Z := 270.122; Lines5[69].F := 1000; Lines5[69].CMD := 2; Lines5[69].Param := 0; // G1 Continuous [Op72 P1]
    Lines5[70].X := 270.914; Lines5[70].Z := 266.690; Lines5[70].F := 1000; Lines5[70].CMD := 2; Lines5[70].Param := 0; // G1 Continuous [Op72 P1]
    Lines5[71].X := 270.367; Lines5[71].Z := 263.243; Lines5[71].F := 1000; Lines5[71].CMD := 2; Lines5[71].Param := 0; // G1 Continuous [Op72 P1]
    Lines5[72].X := 269.765; Lines5[72].Z := 259.784; Lines5[72].F := 1000; Lines5[72].CMD := 2; Lines5[72].Param := 0; // G1 Continuous [Op72 P1]
    Lines5[73].X := 269.110; Lines5[73].Z := 256.317; Lines5[73].F := 1000; Lines5[73].CMD := 2; Lines5[73].Param := 0; // G1 Continuous [Op72 P1]
    Lines5[74].X := 268.337; Lines5[74].Z := 252.531; Lines5[74].F := 1000; Lines5[74].CMD := 2; Lines5[74].Param := 0; // G1 Continuous [Op72 P1]
    Lines5[75].X := 267.577; Lines5[75].Z := 249.061; Lines5[75].F := 1000; Lines5[75].CMD := 2; Lines5[75].Param := 0; // G1 Continuous [Op72 P1]
    Lines5[76].X := 266.695; Lines5[76].Z := 245.281; Lines5[76].F := 1000; Lines5[76].CMD := 2; Lines5[76].Param := 0; // G1 Continuous [Op72 P1]
    Lines5[77].X := 265.759; Lines5[77].Z := 241.511; Lines5[77].F := 1000; Lines5[77].CMD := 2; Lines5[77].Param := 0; // G1 Continuous [Op72 P1]
    Lines5[78].X := 264.774; Lines5[78].Z := 237.756; Lines5[78].F := 1000; Lines5[78].CMD := 2; Lines5[78].Param := 0; // G1 Continuous [Op72 P1]
    Lines5[79].X := 263.741; Lines5[79].Z := 234.022; Lines5[79].F := 1000; Lines5[79].CMD := 2; Lines5[79].Param := 0; // G1 Continuous [Op72 P1]
    Lines5[80].X := 262.663; Lines5[80].Z := 230.314; Lines5[80].F := 1000; Lines5[80].CMD := 2; Lines5[80].Param := 0; // G1 Continuous [Op72 P1]
    Lines5[81].X := 261.544; Lines5[81].Z := 226.636; Lines5[81].F := 1000; Lines5[81].CMD := 2; Lines5[81].Param := 0; // G1 Continuous [Op72 P1]
    Lines5[82].X := 260.287; Lines5[82].Z := 222.693; Lines5[82].F := 1000; Lines5[82].CMD := 2; Lines5[82].Param := 0; // G1 Continuous [Op72 P1]
    Lines5[83].X := 259.089; Lines5[83].Z := 219.096; Lines5[83].F := 1000; Lines5[83].CMD := 2; Lines5[83].Param := 0; // G1 Continuous [Op72 P1]
    Lines5[84].X := 257.753; Lines5[84].Z := 215.251; Lines5[84].F := 1000; Lines5[84].CMD := 2; Lines5[84].Param := 0; // G1 Continuous [Op72 P1]
    Lines5[85].X := 256.382; Lines5[85].Z := 211.468; Lines5[85].F := 1000; Lines5[85].CMD := 2; Lines5[85].Param := 0; // G1 Continuous [Op72 P1]
    Lines5[86].X := 254.978; Lines5[86].Z := 207.752; Lines5[86].F := 1000; Lines5[86].CMD := 2; Lines5[86].Param := 0; // G1 Continuous [Op72 P1]
    Lines5[87].X := 253.546; Lines5[87].Z := 204.110; Lines5[87].F := 1000; Lines5[87].CMD := 2; Lines5[87].Param := 0; // G1 Continuous [Op72 P1]
    Lines5[88].X := 252.088; Lines5[88].Z := 200.548; Lines5[88].F := 1000; Lines5[88].CMD := 2; Lines5[88].Param := 0; // G1 Continuous [Op72 P1]
    Lines5[89].X := 250.609; Lines5[89].Z := 197.073; Lines5[89].F := 1000; Lines5[89].CMD := 2; Lines5[89].Param := 0; // G1 Continuous [Op72 P1]
    Lines5[90].X := 249.111; Lines5[90].Z := 193.691; Lines5[90].F := 1000; Lines5[90].CMD := 2; Lines5[90].Param := 0; // G1 Continuous [Op72 P1]
    Lines5[91].X := 247.599; Lines5[91].Z := 190.410; Lines5[91].F := 1000; Lines5[91].CMD := 2; Lines5[91].Param := 0; // G1 Continuous [Op72 P1]
    Lines5[92].X := 246.075; Lines5[92].Z := 187.234; Lines5[92].F := 1000; Lines5[92].CMD := 2; Lines5[92].Param := 0; // G1 Continuous [Op72 P1]
    Lines5[93].X := 244.544; Lines5[93].Z := 184.171; Lines5[93].F := 1000; Lines5[93].CMD := 2; Lines5[93].Param := 0; // G1 Continuous [Op72 P1]
    Lines5[94].X := 242.890; Lines5[94].Z := 181.006; Lines5[94].F := 1000; Lines5[94].CMD := 2; Lines5[94].Param := 0; // G1 Continuous [Op72 P1]
    Lines5[95].X := 242.890; Lines5[95].Z := 74.000; Lines5[95].F := 0; Lines5[95].CMD := 0; Lines5[95].Param := 0; // G0 Rapid [Op72 P1]
    Lines5[96].X := 174.000; Lines5[96].Z := 74.000; Lines5[96].F := 0; Lines5[96].CMD := 0; Lines5[96].Param := 0; // G0 Rapid [Op72 P1]
    Lines5[97].X := 174.000; Lines5[97].Z := 74.000; Lines5[97].F := 0; Lines5[97].CMD := 21; Lines5[97].Param := 0; // Spindle OFF [Op72 P1]
    Lines5[98].X := 174.000; Lines5[98].Z := 74.000; Lines5[98].F := 0; Lines5[98].CMD := 21; Lines5[98].Param := 0; // Spindle OFF
    Lines5[99].X := 0.000; Lines5[99].Z := 0.000; Lines5[99].F := 0; Lines5[99].CMD := 99; Lines5[99].Param := 0; // Program END
END_DATA_BLOCK